LIN {X 0,Y 573.745,Z 549.18,A -85,B 0,C 180,E1 -2261.974,E2 -2261.974} C_VEL
LIN {X 0,Y 573.825,Z 536.531,A -85,B 0,C 180,E1 -2262.331,E2 -2262.331} C_VEL
LIN {X 0,Y 573.935,Z 523.333,A -85,B 0,C 180,E1 -2262.553,E2 -2262.553} C_VEL
LIN {X 0,Y 573.912,Z 426.198,A -85,B 0,C 180,E1 -2263.777,E2 -2263.777} C_VEL
LIN {X 0,Y 573.403,Z 422.615,A -85,B 0,C 180,E1 -2263.85,E2 -2263.85} C_VEL
LIN {X 0,Y 573.571,Z 402.121,A -85,B 0,C 180,E1 -2266.727,E2 -2266.727} C_VEL
LIN {X 0,Y 573.815,Z 381.614,A -85,B 0,C 180,E1 -2269.645,E2 -2269.645} C_VEL
LIN {X 0,Y 574.108,Z 361.938,A -85,B 0,C 180,E1 -2272.491,E2 -2272.491} C_VEL
LIN {X 0,Y 573.627,Z 356.944,A -85,B 0,C 180,E1 -2273.235,E2 -2273.235} C_VEL
LIN {X 0,Y 573.261,Z 355.081,A -85,B 0,C 180,E1 -2273.543,E2 -2273.543} C_VEL
LIN {X 0,Y 573.265,Z 355.076,A -85,B 0,C 180,E1 -2276.189,E2 -2276.189} C_VEL
LIN {X 0,Y 573.239,Z 355.076,A -85,B 0,C 180,E1 -2278.564,E2 -2278.564} C_VEL
LIN {X 0,Y 573.235,Z 355.076,A -85,B 0,C 180,E1 -2280.992,E2 -2280.992} C_VEL
LIN {X 0,Y 573.261,Z 355.078,A -85,B 0,C 180,E1 -2283.523,E2 -2283.523} C_VEL
LIN {X 0,Y 573.26,Z 355.076,A -85,B 0,C 180,E1 -2286.047,E2 -2286.047} C_VEL
LIN {X 0,Y 573.247,Z 355.073,A -85,B 0,C 180,E1 -2288.7,E2 -2288.7} C_VEL
LIN {X 0,Y 573.251,Z 355.083,A -85,B 0,C 180,E1 -2291.595,E2 -2291.595} C_VEL
LIN {X 0,Y 573.235,Z 355.075,A -85,B 0,C 180,E1 -2294.332,E2 -2294.332} C_VEL
LIN {X 0,Y 573.247,Z 355.08,A -85,B 0,C 180,E1 -2297.356,E2 -2297.356} C_VEL
LIN {X 0,Y 573.245,Z 355.073,A -85,B 0,C 180,E1 -2300.393,E2 -2300.393} C_VEL
LIN {X 0,Y 573.251,Z 355.077,A -85,B 0,C 180,E1 -2303.077,E2 -2303.077} C_VEL
LIN {X 0,Y 573.268,Z 355.076,A -85,B 0,C 180,E1 -2305.671,E2 -2305.671} C_VEL
LIN {X 0,Y 573.245,Z 355.074,A -85,B 0,C 180,E1 -2308.185,E2 -2308.185} C_VEL
LIN {X 0,Y 573.264,Z 355.072,A -85,B 0,C 180,E1 -2310.634,E2 -2310.634} C_VEL
LIN {X 0,Y 573.265,Z 355.078,A -85,B 0,C 180,E1 -2313.499,E2 -2313.499} C_VEL
LIN {X 0,Y 573.237,Z 355.074,A -85,B 0,C 180,E1 -2316.135,E2 -2316.135} C_VEL
LIN {X 0,Y 573.252,Z 355.075,A -85,B 0,C 180,E1 -2318.706,E2 -2318.706} C_VEL
LIN {X 0,Y 573.233,Z 355.081,A -85,B 0,C 180,E1 -2321.412,E2 -2321.412} C_VEL
LIN {X 0,Y 573.253,Z 355.075,A -85,B 0,C 180,E1 -2323.622,E2 -2323.622} C_VEL
LIN {X 0,Y 573.232,Z 355.077,A -85,B 0,C 180,E1 -2326.529,E2 -2326.529} C_VEL
LIN {X 0,Y 573.269,Z 355.075,A -85,B 0,C 180,E1 -2329.403,E2 -2329.403} C_VEL
LIN {X 0,Y 573.282,Z 355.069,A -85,B 0,C 180,E1 -2332.25,E2 -2332.25} C_VEL
LIN {X 0,Y 573.308,Z 355.075,A -85,B 0,C 180,E1 -2335.077,E2 -2335.077} C_VEL
LIN {X 0,Y 573.301,Z 355.066,A -85,B 0,C 180,E1 -2337.892,E2 -2337.892} C_VEL
LIN {X 0,Y 573.333,Z 355.069,A -85,B 0,C 180,E1 -2340.702,E2 -2340.702} C_VEL
LIN {X 0,Y 573.238,Z 355.076,A -85,B 0,C 180,E1 -2343.515,E2 -2343.515} C_VEL
LIN {X 0,Y 573.287,Z 355.069,A -85,B 0,C 180,E1 -2345.628,E2 -2345.628} C_VEL
LIN {X 0,Y 573.3,Z 355.071,A -85,B 0,C 180,E1 -2348.459,E2 -2348.459} C_VEL
LIN {X 0,Y 573.29,Z 355.07,A -85,B 0,C 180,E1 -2351.312,E2 -2351.312} C_VEL
LIN {X 0,Y 573.272,Z 355.075,A -85,B 0,C 180,E1 -2354.425,E2 -2354.425} C_VEL
LIN {X 0,Y 573.253,Z 355.076,A -85,B 0,C 180,E1 -2357.112,E2 -2357.112} C_VEL
LIN {X 0,Y 573.251,Z 355.074,A -85,B 0,C 180,E1 -2360.077,E2 -2360.077} C_VEL
LIN {X 0,Y 573.264,Z 355.073,A -85,B 0,C 180,E1 -2363.154,E2 -2363.154} C_VEL
LIN {X 0,Y 573.247,Z 355.079,A -85,B 0,C 180,E1 -2364.408,E2 -2364.408} C_VEL
LIN {X 0,Y 572.616,Z 355.163,A -85,B 0,C 180,E1 -2364.994,E2 -2364.994} C_VEL
LIN {X 0,Y 569.776,Z 355.516,A -85,B 0,C 180,E1 -2365.946,E2 -2365.946} C_VEL
LIN {X 0,Y 567.349,Z 355.816,A -85,B 0,C 180,E1 -2366.712,E2 -2366.712} C_VEL
LIN {X 0,Y 566.298,Z 355.94,A -85,B 0,C 180,E1 -2367.303,E2 -2367.303} C_VEL
LIN {X 0,Y 566.21,Z 355.95,A -85,B 0,C 180,E1 -2367.503,E2 -2367.503} C_VEL
LIN {X 0,Y 566.182,Z 355.962,A -85,B 0,C 180,E1 -2370.593,E2 -2370.593} C_VEL
LIN {X 0,Y 566.223,Z 355.95,A -85,B 0,C 180,E1 -2373.102,E2 -2373.102} C_VEL
LIN {X 0,Y 566.2,Z 355.957,A -85,B 0,C 180,E1 -2376.216,E2 -2376.216} C_VEL
LIN {X 0,Y 566.216,Z 355.949,A -85,B 0,C 180,E1 -2379.274,E2 -2379.274} C_VEL
LIN {X 0,Y 566.212,Z 355.955,A -85,B 0,C 180,E1 -2382.088,E2 -2382.088} C_VEL
LIN {X 0,Y 566.169,Z 355.956,A -85,B 0,C 180,E1 -2385.037,E2 -2385.037} C_VEL
LIN {X 0,Y 566.186,Z 355.957,A -85,B 0,C 180,E1 -2387.911,E2 -2387.911} C_VEL
LIN {X 0,Y 566.22,Z 355.951,A -85,B 0,C 180,E1 -2390.728,E2 -2390.728} C_VEL
LIN {X 0,Y 566.217,Z 355.952,A -85,B 0,C 180,E1 -2393.784,E2 -2393.784} C_VEL
LIN {X 0,Y 566.212,Z 355.958,A -85,B 0,C 180,E1 -2396.266,E2 -2396.266} C_VEL
LIN {X 0,Y 566.198,Z 355.952,A -85,B 0,C 180,E1 -2398.923,E2 -2398.923} C_VEL
LIN {X 0,Y 566.212,Z 355.955,A -85,B 0,C 180,E1 -2401.858,E2 -2401.858} C_VEL
LIN {X 0,Y 566.215,Z 355.957,A -85,B 0,C 180,E1 -2404.252,E2 -2404.252} C_VEL
LIN {X 0,Y 566.171,Z 355.957,A -85,B 0,C 180,E1 -2406.72,E2 -2406.72} C_VEL
LIN {X 0,Y 566.209,Z 355.956,A -85,B 0,C 180,E1 -2409.663,E2 -2409.663} C_VEL
LIN {X 0,Y 566.264,Z 356.15,A -85,B 0,C 180,E1 -2410.878,E2 -2410.878} C_VEL
LIN {X 0,Y 566.436,Z 363.825,A -85,B 0,C 180,E1 -2412.304,E2 -2412.304} C_VEL
LIN {X 0,Y 566.321,Z 379.961,A -85,B 0,C 180,E1 -2415.249,E2 -2415.249} C_VEL
LIN {X 0,Y 566.257,Z 384.42,A -85,B 0,C 180,E1 -2416.055,E2 -2416.055} C_VEL
LIN {X 0,Y 567.176,Z 390.378,A -85,B 0,C 180,E1 -2416.155,E2 -2416.155} C_VEL
LIN {X 0,Y 566.94,Z 490.984,A -85,B 0,C 180,E1 -2417.448,E2 -2417.448} C_VEL
LIN {X 0,Y 566.86,Z 504.235,A -85,B 0,C 180,E1 -2417.765,E2 -2417.765} C_VEL
LIN {X 0,Y 566.745,Z 516.388,A -85,B 0,C 180,E1 -2418.194,E2 -2418.194} C_VEL
LIN {X 0,Y 566.619,Z 528.384,A -85,B 0,C 180,E1 -2418.766,E2 -2418.766} C_VEL
LIN {X 0,Y 566.464,Z 539.56,A -85,B 0,C 180,E1 -2419.456,E2 -2419.456} C_VEL
LIN {X 0,Y 566.326,Z 550.076,A -85,B 0,C 180,E1 -2420.266,E2 -2420.266} C_VEL
LIN {X 0,Y 566.221,Z 558.671,A -85,B 0,C 180,E1 -2421.075,E2 -2421.075} C_VEL
LIN {X 0,Y 566.113,Z 566.592,A -85,B 0,C 180,E1 -2421.972,E2 -2421.972} C_VEL
LIN {X 0,Y 566.05,Z 573.16,A -85,B 0,C 180,E1 -2422.868,E2 -2422.868} C_VEL
LIN {X 0,Y 566.003,Z 579.628,A -85,B 0,C 180,E1 -2423.942,E2 -2423.942} C_VEL
LIN {X 0,Y 565.878,Z 584.765,A -85,B 0,C 180,E1 -2425.013,E2 -2425.013} C_VEL
LIN {X 0,Y 565.926,Z 588.754,A -85,B 0,C 180,E1 -2426.084,E2 -2426.084} C_VEL
LIN {X 0,Y 565.877,Z 591.702,A -85,B 0,C 180,E1 -2427.153,E2 -2427.153} C_VEL
LIN {X 0,Y 565.84,Z 593.128,A -85,B 0,C 180,E1 -2427.865,E2 -2427.865} C_VEL
LIN {X 0,Y 565.841,Z 594.756,A -85,B 0,C 180,E1 -2429.288,E2 -2429.288} C_VEL
LIN {X 0,Y 565.839,Z 594.996,A -85,B 0,C 180,E1 -2430,E2 -2430} C_VEL
LIN {X 0,Y 565.841,Z 594.815,A -85,B 0,C 180,E1 -2430.712,E2 -2430.712} C_VEL
LIN {X 0,Y 565.841,Z 593.268,A -85,B 0,C 180,E1 -2432.135,E2 -2432.135} C_VEL
LIN {X 0,Y 565.878,Z 591.907,A -85,B 0,C 180,E1 -2432.847,E2 -2432.847} C_VEL
LIN {X 0,Y 565.927,Z 589.03,A -85,B 0,C 180,E1 -2433.916,E2 -2433.916} C_VEL
LIN {X 0,Y 565.878,Z 585.13,A -85,B 0,C 180,E1 -2434.987,E2 -2434.987} C_VEL
LIN {X 0,Y 565.99,Z 580.097,A -85,B 0,C 180,E1 -2436.058,E2 -2436.058} C_VEL
LIN {X 0,Y 566.031,Z 573.773,A -85,B 0,C 180,E1 -2437.132,E2 -2437.132} C_VEL
LIN {X 0,Y 566.128,Z 565.852,A -85,B 0,C 180,E1 -2438.208,E2 -2438.208} C_VEL
LIN {X 0,Y 566.249,Z 556.001,A -85,B 0,C 180,E1 -2439.285,E2 -2439.285} C_VEL
LIN {X 0,Y 566.42,Z 545.683,A -85,B 0,C 180,E1 -2440.184,E2 -2440.184} C_VEL
LIN {X 0,Y 566.56,Z 534.375,A -85,B 0,C 180,E1 -2440.973,E2 -2440.973} C_VEL
LIN {X 0,Y 566.691,Z 523.193,A -85,B 0,C 180,E1 -2441.592,E2 -2441.592} C_VEL
LIN {X 0,Y 566.794,Z 510.602,A -85,B 0,C 180,E1 -2442.119,E2 -2442.119} C_VEL
LIN {X 0,Y 566.876,Z 497.43,A -85,B 0,C 180,E1 -2442.508,E2 -2442.508} C_VEL
LIN {X 0,Y 566.978,Z 485.069,A -85,B 0,C 180,E1 -2442.733,E2 -2442.733} C_VEL
LIN {X 0,Y 567.07,Z 389.372,A -85,B 0,C 180,E1 -2443.951,E2 -2443.951} C_VEL
LIN {X 0,Y 566.252,Z 384.332,A -85,B 0,C 180,E1 -2444.051,E2 -2444.051} C_VEL
LIN {X 0,Y 566.417,Z 367.153,A -85,B 0,C 180,E1 -2447.175,E2 -2447.175} C_VEL
LIN {X 0,Y 566.346,Z 356.612,A -85,B 0,C 180,E1 -2449.123,E2 -2449.123} C_VEL
LIN {X 0,Y 566.235,Z 355.953,A -85,B 0,C 180,E1 -2449.295,E2 -2449.295} C_VEL
LIN {X 0,Y 566.197,Z 355.961,A -85,B 0,C 180,E1 -2451.862,E2 -2451.862} C_VEL
LIN {X 0,Y 566.238,Z 355.948,A -85,B 0,C 180,E1 -2454.96,E2 -2454.96} C_VEL
LIN {X 0,Y 566.212,Z 355.951,A -85,B 0,C 180,E1 -2457.338,E2 -2457.338} C_VEL
LIN {X 0,Y 566.203,Z 355.957,A -85,B 0,C 180,E1 -2459.768,E2 -2459.768} C_VEL
LIN {X 0,Y 566.206,Z 355.953,A -85,B 0,C 180,E1 -2462.43,E2 -2462.43} C_VEL
LIN {X 0,Y 566.213,Z 355.949,A -85,B 0,C 180,E1 -2464.994,E2 -2464.994} C_VEL
LIN {X 0,Y 566.195,Z 355.955,A -85,B 0,C 180,E1 -2467.46,E2 -2467.46} C_VEL
LIN {X 0,Y 566.225,Z 355.952,A -85,B 0,C 180,E1 -2470.196,E2 -2470.196} C_VEL
LIN {X 0,Y 566.197,Z 355.952,A -85,B 0,C 180,E1 -2473.053,E2 -2473.053} C_VEL
LIN {X 0,Y 566.198,Z 355.956,A -85,B 0,C 180,E1 -2476.047,E2 -2476.047} C_VEL
LIN {X 0,Y 566.207,Z 355.95,A -85,B 0,C 180,E1 -2478.863,E2 -2478.863} C_VEL
LIN {X 0,Y 566.185,Z 355.963,A -85,B 0,C 180,E1 -2481.637,E2 -2481.637} C_VEL
LIN {X 0,Y 566.206,Z 355.951,A -85,B 0,C 180,E1 -2484.311,E2 -2484.311} C_VEL
LIN {X 0,Y 566.223,Z 355.949,A -85,B 0,C 180,E1 -2486.898,E2 -2486.898} C_VEL
LIN {X 0,Y 566.182,Z 355.961,A -85,B 0,C 180,E1 -2489.407,E2 -2489.407} C_VEL
LIN {X 0,Y 566.221,Z 355.953,A -85,B 0,C 180,E1 -2491.858,E2 -2491.858} C_VEL
LIN {X 0,Y 566.217,Z 355.949,A -85,B 0,C 180,E1 -2494.251,E2 -2494.251} C_VEL
LIN {X 0,Y 566.196,Z 355.961,A -85,B 0,C 180,E1 -2497.369,E2 -2497.369} C_VEL
LIN {X 0,Y 566.213,Z 355.955,A -85,B 0,C 180,E1 -2499.663,E2 -2499.663} C_VEL
LIN {X 0,Y 566.197,Z 355.952,A -85,B 0,C 180,E1 -2502.668,E2 -2502.668} C_VEL
LIN {X 0,Y 566.224,Z 355.953,A -85,B 0,C 180,E1 -2505.626,E2 -2505.626} C_VEL
LIN {X 0,Y 566.266,Z 355.944,A -85,B 0,C 180,E1 -2508.654,E2 -2508.654} C_VEL
LIN {X 0,Y 566.241,Z 355.952,A -85,B 0,C 180,E1 -2511.434,E2 -2511.434} C_VEL
LIN {X 0,Y 566.254,Z 355.944,A -85,B 0,C 180,E1 -2514.302,E2 -2514.302} C_VEL
LIN {X 0,Y 566.273,Z 355.943,A -85,B 0,C 180,E1 -2517.866,E2 -2517.866} C_VEL
LIN {X 0,Y 566.301,Z 355.942,A -85,B 0,C 180,E1 -2520.711,E2 -2520.711} C_VEL
LIN {X 0,Y 566.274,Z 355.948,A -85,B 0,C 180,E1 -2522.846,E2 -2522.846} C_VEL
LIN {X 0,Y 566.255,Z 355.945,A -85,B 0,C 180,E1 -2525.698,E2 -2525.698} C_VEL
LIN {X 0,Y 566.242,Z 355.949,A -85,B 0,C 180,E1 -2528.565,E2 -2528.565} C_VEL
LIN {X 0,Y 566.242,Z 355.948,A -85,B 0,C 180,E1 -2531.454,E2 -2531.454} C_VEL
LIN {X 0,Y 566.225,Z 355.952,A -85,B 0,C 180,E1 -2534.507,E2 -2534.507} C_VEL
LIN {X 0,Y 566.197,Z 355.954,A -85,B 0,C 180,E1 -2537.332,E2 -2537.332} C_VEL
LIN {X 0,Y 566.216,Z 355.952,A -85,B 0,C 180,E1 -2540.337,E2 -2540.337} C_VEL
LIN {X 0,Y 566.222,Z 355.95,A -85,B 0,C 180,E1 -2543.402,E2 -2543.402} C_VEL
LIN {X 0,Y 566.218,Z 355.949,A -85,B 0,C 180,E1 -2545.749,E2 -2545.749} C_VEL
LIN {X 0,Y 566.202,Z 355.953,A -85,B 0,C 180,E1 -2548.204,E2 -2548.204} C_VEL
LIN {X 0,Y 566.194,Z 355.955,A -85,B 0,C 180,E1 -2551.079,E2 -2551.079} C_VEL
LIN {X 0,Y 566.223,Z 355.948,A -85,B 0,C 180,E1 -2553.738,E2 -2553.738} C_VEL
LIN {X 0,Y 566.211,Z 355.96,A -85,B 0,C 180,E1 -2556.569,E2 -2556.569} C_VEL
LIN {X 0,Y 566.209,Z 355.95,A -85,B 0,C 180,E1 -2559.687,E2 -2559.687} C_VEL
LIN {X 0,Y 566.213,Z 355.953,A -85,B 0,C 180,E1 -2562.088,E2 -2562.088} C_VEL
LIN {X 0,Y 566.17,Z 355.957,A -85,B 0,C 180,E1 -2565.036,E2 -2565.036} C_VEL
LIN {X 0,Y 566.215,Z 355.954,A -85,B 0,C 180,E1 -2568.137,E2 -2568.137} C_VEL
LIN {X 0,Y 566.22,Z 355.953,A -85,B 0,C 180,E1 -2570.728,E2 -2570.728} C_VEL
LIN {X 0,Y 566.217,Z 355.951,A -85,B 0,C 180,E1 -2573.784,E2 -2573.784} C_VEL
LIN {X 0,Y 566.211,Z 355.959,A -85,B 0,C 180,E1 -2576.266,E2 -2576.266} C_VEL
LIN {X 0,Y 566.198,Z 355.952,A -85,B 0,C 180,E1 -2578.923,E2 -2578.923} C_VEL
LIN {X 0,Y 566.211,Z 355.955,A -85,B 0,C 180,E1 -2581.858,E2 -2581.858} C_VEL
LIN {X 0,Y 566.215,Z 355.959,A -85,B 0,C 180,E1 -2584.252,E2 -2584.252} C_VEL
LIN {X 0,Y 566.236,Z 356.138,A -85,B 0,C 180,E1 -2586.356,E2 -2586.356} C_VEL
LIN {X 0,Y 567.11,Z 361.752,A -85,B 0,C 180,E1 -2587.216,E2 -2587.216} C_VEL
LIN {X 0,Y 566.912,Z 380.06,A -85,B 0,C 180,E1 -2589.879,E2 -2589.879} C_VEL
LIN {X 0,Y 566.61,Z 400.895,A -85,B 0,C 180,E1 -2592.885,E2 -2592.885} C_VEL
LIN {X 0,Y 566.403,Z 422.615,A -85,B 0,C 180,E1 -2595.975,E2 -2595.975} C_VEL
LIN {X 0,Y 567.22,Z 429.316,A -85,B 0,C 180,E1 -2596.097,E2 -2596.097} C_VEL
LIN {X 0,Y 566.937,Z 530.961,A -85,B 0,C 180,E1 -2597.403,E2 -2597.403} C_VEL
LIN {X 0,Y 566.859,Z 544.228,A -85,B 0,C 180,E1 -2597.719,E2 -2597.719} C_VEL
LIN {X 0,Y 566.758,Z 556.383,A -85,B 0,C 180,E1 -2598.149,E2 -2598.149} C_VEL
LIN {X 0,Y 566.589,Z 568.447,A -85,B 0,C 180,E1 -2598.724,E2 -2598.724} C_VEL
LIN {X 0,Y 566.442,Z 580.203,A -85,B 0,C 180,E1 -2599.455,E2 -2599.455} C_VEL
LIN {X 0,Y 566.321,Z 590.605,A -85,B 0,C 180,E1 -2600.266,E2 -2600.266} C_VEL
LIN {X 0,Y 566.207,Z 599.115,A -85,B 0,C 180,E1 -2601.074,E2 -2601.074} C_VEL
LIN {X 0,Y 566.112,Z 606.962,A -85,B 0,C 180,E1 -2601.972,E2 -2601.972} C_VEL
LIN {X 0,Y 566.003,Z 614.623,A -85,B 0,C 180,E1 -2603.047,E2 -2603.047} C_VEL
LIN {X 0,Y 566.004,Z 621.68,A -85,B 0,C 180,E1 -2604.299,E2 -2604.299} C_VEL
LIN {X 0,Y 565.933,Z 626.373,A -85,B 0,C 180,E1 -2605.37,E2 -2605.37} C_VEL
LIN {X 0,Y 565.927,Z 629.958,A -85,B 0,C 180,E1 -2606.44,E2 -2606.44} C_VEL
LIN {X 0,Y 565.878,Z 631.808,A -85,B 0,C 180,E1 -2607.153,E2 -2607.153} C_VEL
LIN {X 0,Y 565.846,Z 634.185,A -85,B 0,C 180,E1 -2608.577,E2 -2608.577} C_VEL
LIN {X 0,Y 565.839,Z 635,A -85,B 0,C 180,E1 -2610,E2 -2610} C_VEL
LIN {X 0,Y 565.846,Z 634.186,A -85,B 0,C 180,E1 -2611.423,E2 -2611.423} C_VEL
LIN {X 0,Y 565.878,Z 631.81,A -85,B 0,C 180,E1 -2612.847,E2 -2612.847} C_VEL
LIN {X 0,Y 565.926,Z 628.896,A -85,B 0,C 180,E1 -2613.916,E2 -2613.916} C_VEL
LIN {X 0,Y 565.878,Z 624.949,A -85,B 0,C 180,E1 -2614.987,E2 -2614.987} C_VEL
LIN {X 0,Y 566.002,Z 619.868,A -85,B 0,C 180,E1 -2616.058,E2 -2616.058} C_VEL
LIN {X 0,Y 566.04,Z 613.469,A -85,B 0,C 180,E1 -2617.132,E2 -2617.132} C_VEL
LIN {X 0,Y 566.133,Z 605.479,A -85,B 0,C 180,E1 -2618.207,E2 -2618.207} C_VEL
LIN {X 0,Y 566.228,Z 597.337,A -85,B 0,C 180,E1 -2619.105,E2 -2619.105} C_VEL
LIN {X 0,Y 566.343,Z 587.403,A -85,B 0,C 180,E1 -2620.005,E2 -2620.005} C_VEL
LIN {X 0,Y 566.529,Z 576.294,A -85,B 0,C 180,E1 -2620.807,E2 -2620.807} C_VEL
LIN {X 0,Y 566.612,Z 565.181,A -85,B 0,C 180,E1 -2621.446,E2 -2621.446} C_VEL
LIN {X 0,Y 566.736,Z 552.989,A -85,B 0,C 180,E1 -2621.988,E2 -2621.988} C_VEL
LIN {X 0,Y 566.892,Z 540.187,A -85,B 0,C 180,E1 -2622.394,E2 -2622.394} C_VEL
LIN {X 0,Y 567.001,Z 528.125,A -85,B 0,C 180,E1 -2622.641,E2 -2622.641} C_VEL
LIN {X 0,Y 567.055,Z 427.203,A -85,B 0,C 180,E1 -2623.934,E2 -2623.934} C_VEL
LIN {X 0,Y 566.403,Z 422.615,A -85,B 0,C 180,E1 -2624.025,E2 -2624.025} C_VEL
LIN {X 0,Y 566.61,Z 400.895,A -85,B 0,C 180,E1 -2627.115,E2 -2627.115} C_VEL
LIN {X 0,Y 566.912,Z 380.062,A -85,B 0,C 180,E1 -2630.121,E2 -2630.121} C_VEL
LIN {X 0,Y 567.109,Z 361.752,A -85,B 0,C 180,E1 -2632.784,E2 -2632.784} C_VEL
LIN {X 0,Y 566.22,Z 355.959,A -85,B 0,C 180,E1 -2633.693,E2 -2633.693} C_VEL
LIN {X 0,Y 566.216,Z 355.95,A -85,B 0,C 180,E1 -2636.54,E2 -2636.54} C_VEL
LIN {X 0,Y 566.193,Z 355.953,A -85,B 0,C 180,E1 -2638.953,E2 -2638.953} C_VEL
LIN {X 0,Y 566.2,Z 355.957,A -85,B 0,C 180,E1 -2641.421,E2 -2641.421} C_VEL
LIN {X 0,Y 566.212,Z 355.955,A -85,B 0,C 180,E1 -2643.955,E2 -2643.955} C_VEL
LIN {X 0,Y 566.215,Z 355.949,A -85,B 0,C 180,E1 -2646.568,E2 -2646.568} C_VEL
LIN {X 0,Y 566.211,Z 355.959,A -85,B 0,C 180,E1 -2649.685,E2 -2649.685} C_VEL
LIN {X 0,Y 566.211,Z 355.952,A -85,B 0,C 180,E1 -2652.086,E2 -2652.086} C_VEL
LIN {X 0,Y 566.17,Z 355.957,A -85,B 0,C 180,E1 -2655.035,E2 -2655.035} C_VEL
LIN {X 0,Y 566.213,Z 355.953,A -85,B 0,C 180,E1 -2657.912,E2 -2657.912} C_VEL
LIN {X 0,Y 566.218,Z 355.949,A -85,B 0,C 180,E1 -2660.726,E2 -2660.726} C_VEL
LIN {X 0,Y 566.212,Z 355.954,A -85,B 0,C 180,E1 -2663.783,E2 -2663.783} C_VEL
LIN {X 0,Y 566.223,Z 355.948,A -85,B 0,C 180,E1 -2666.262,E2 -2666.262} C_VEL
LIN {X 0,Y 566.197,Z 355.954,A -85,B 0,C 180,E1 -2668.921,E2 -2668.921} C_VEL
LIN {X 0,Y 566.192,Z 355.957,A -85,B 0,C 180,E1 -2671.047,E2 -2671.047} C_VEL
LIN {X 0,Y 566.24,Z 355.953,A -85,B 0,C 180,E1 -2673.46,E2 -2673.46} C_VEL
LIN {X 0,Y 566.197,Z 355.953,A -85,B 0,C 180,E1 -2675.819,E2 -2675.819} C_VEL
LIN {X 0,Y 566.211,Z 355.954,A -85,B 0,C 180,E1 -2678.902,E2 -2678.902} C_VEL
LIN {X 0,Y 566.206,Z 355.96,A -85,B 0,C 180,E1 -2681.172,E2 -2681.172} C_VEL
LIN {X 0,Y 566.215,Z 355.955,A -85,B 0,C 180,E1 -2683.412,E2 -2683.412} C_VEL
LIN {X 0,Y 566.194,Z 355.952,A -85,B 0,C 180,E1 -2686.359,E2 -2686.359} C_VEL
LIN {X 0,Y 566.266,Z 355.946,A -85,B 0,C 180,E1 -2688.654,E2 -2688.654} C_VEL
LIN {X 0,Y 566.241,Z 355.95,A -85,B 0,C 180,E1 -2691.434,E2 -2691.434} C_VEL
LIN {X 0,Y 566.255,Z 355.945,A -85,B 0,C 180,E1 -2694.302,E2 -2694.302} C_VEL
LIN {X 0,Y 566.273,Z 355.942,A -85,B 0,C 180,E1 -2697.866,E2 -2697.866} C_VEL
LIN {X 0,Y 566.303,Z 355.944,A -85,B 0,C 180,E1 -2700.711,E2 -2700.711} C_VEL
LIN {X 0,Y 566.274,Z 355.951,A -85,B 0,C 180,E1 -2702.846,E2 -2702.846} C_VEL
LIN {X 0,Y 566.255,Z 355.944,A -85,B 0,C 180,E1 -2705.698,E2 -2705.698} C_VEL
LIN {X 0,Y 566.241,Z 355.951,A -85,B 0,C 180,E1 -2708.566,E2 -2708.566} C_VEL
LIN {X 0,Y 566.242,Z 355.947,A -85,B 0,C 180,E1 -2711.454,E2 -2711.454} C_VEL
LIN {X 0,Y 566.225,Z 355.954,A -85,B 0,C 180,E1 -2714.507,E2 -2714.507} C_VEL
LIN {X 0,Y 566.197,Z 355.953,A -85,B 0,C 180,E1 -2717.332,E2 -2717.332} C_VEL
LIN {X 0,Y 566.213,Z 355.954,A -85,B 0,C 180,E1 -2720.337,E2 -2720.337} C_VEL
LIN {X 0,Y 566.222,Z 355.949,A -85,B 0,C 180,E1 -2723.403,E2 -2723.403} C_VEL
LIN {X 0,Y 566.218,Z 355.949,A -85,B 0,C 180,E1 -2725.749,E2 -2725.749} C_VEL
LIN {X 0,Y 566.21,Z 355.95,A -85,B 0,C 180,E1 -2727.503,E2 -2727.503} C_VEL
LIN {X 0,Y 565.53,Z 356.039,A -85,B 0,C 180,E1 -2728.097,E2 -2728.097} C_VEL
LIN {X 0,Y 562.659,Z 356.394,A -85,B 0,C 180,E1 -2729.061,E2 -2729.061} C_VEL
LIN {X 0,Y 560.245,Z 356.695,A -85,B 0,C 180,E1 -2729.836,E2 -2729.836} C_VEL
LIN {X 0,Y 559.218,Z 356.829,A -85,B 0,C 180,E1 -2730.435,E2 -2730.435} C_VEL
LIN {X 0,Y 559.139,Z 356.832,A -85,B 0,C 180,E1 -2730.637,E2 -2730.637} C_VEL
LIN {X 0,Y 559.158,Z 356.828,A -85,B 0,C 180,E1 -2733.575,E2 -2733.575} C_VEL
LIN {X 0,Y 559.177,Z 356.836,A -85,B 0,C 180,E1 -2736.451,E2 -2736.451} C_VEL
LIN {X 0,Y 559.173,Z 356.829,A -85,B 0,C 180,E1 -2738.935,E2 -2738.935} C_VEL
LIN {X 0,Y 559.188,Z 356.826,A -85,B 0,C 180,E1 -2741.768,E2 -2741.768} C_VEL
LIN {X 0,Y 559.136,Z 356.834,A -85,B 0,C 180,E1 -2744.74,E2 -2744.74} C_VEL
LIN {X 0,Y 559.154,Z 356.829,A -85,B 0,C 180,E1 -2747.257,E2 -2747.257} C_VEL
LIN {X 0,Y 559.179,Z 356.833,A -85,B 0,C 180,E1 -2750.136,E2 -2750.136} C_VEL
LIN {X 0,Y 559.145,Z 356.831,A -85,B 0,C 180,E1 -2752.893,E2 -2752.893} C_VEL
LIN {X 0,Y 559.156,Z 356.83,A -85,B 0,C 180,E1 -2755.557,E2 -2755.557} C_VEL
LIN {X 0,Y 559.169,Z 356.837,A -85,B 0,C 180,E1 -2758.138,E2 -2758.138} C_VEL
LIN {X 0,Y 559.144,Z 356.832,A -85,B 0,C 180,E1 -2760.647,E2 -2760.647} C_VEL
LIN {X 0,Y 559.171,Z 356.827,A -85,B 0,C 180,E1 -2763.173,E2 -2763.173} C_VEL
LIN {X 0,Y 559.157,Z 356.832,A -85,B 0,C 180,E1 -2765.496,E2 -2765.496} C_VEL
LIN {X 0,Y 559.173,Z 356.83,A -85,B 0,C 180,E1 -2768.624,E2 -2768.624} C_VEL
LIN {X 0,Y 559.235,Z 357.029,A -85,B 0,C 180,E1 -2770.767,E2 -2770.767} C_VEL
LIN {X 0,Y 559.511,Z 363.855,A -85,B 0,C 180,E1 -2772.077,E2 -2772.077} C_VEL
LIN {X 0,Y 559.276,Z 380.241,A -85,B 0,C 180,E1 -2775.109,E2 -2775.109} C_VEL
LIN {X 0,Y 559.214,Z 384.423,A -85,B 0,C 180,E1 -2775.875,E2 -2775.875} C_VEL
LIN {X 0,Y 560.313,Z 391.886,A -85,B 0,C 180,E1 -2776.001,E2 -2776.001} C_VEL
LIN {X 0,Y 560.026,Z 491.013,A -85,B 0,C 180,E1 -2777.291,E2 -2777.291} C_VEL
LIN {X 0,Y 559.917,Z 504.253,A -85,B 0,C 180,E1 -2777.611,E2 -2777.611} C_VEL
LIN {X 0,Y 559.791,Z 516.403,A -85,B 0,C 180,E1 -2778.045,E2 -2778.045} C_VEL
LIN {X 0,Y 559.656,Z 528.029,A -85,B 0,C 180,E1 -2778.604,E2 -2778.604} C_VEL
LIN {X 0,Y 559.476,Z 539.567,A -85,B 0,C 180,E1 -2779.322,E2 -2779.322} C_VEL
LIN {X 0,Y 559.307,Z 550.083,A -85,B 0,C 180,E1 -2780.142,E2 -2780.142} C_VEL
LIN {X 0,Y 559.197,Z 558.677,A -85,B 0,C 180,E1 -2780.962,E2 -2780.962} C_VEL
LIN {X 0,Y 559.05,Z 566.597,A -85,B 0,C 180,E1 -2781.87,E2 -2781.87} C_VEL
LIN {X 0,Y 558.971,Z 574.457,A -85,B 0,C 180,E1 -2782.977,E2 -2782.977} C_VEL
LIN {X 0,Y 558.936,Z 581.455,A -85,B 0,C 180,E1 -2784.227,E2 -2784.227} C_VEL
LIN {X 0,Y 558.827,Z 586.195,A -85,B 0,C 180,E1 -2785.311,E2 -2785.311} C_VEL
LIN {X 0,Y 558.836,Z 589.828,A -85,B 0,C 180,E1 -2786.395,E2 -2786.395} C_VEL
LIN {X 0,Y 558.799,Z 591.704,A -85,B 0,C 180,E1 -2787.116,E2 -2787.116} C_VEL
LIN {X 0,Y 558.746,Z 593.128,A -85,B 0,C 180,E1 -2787.838,E2 -2787.838} C_VEL
LIN {X 0,Y 558.741,Z 594.757,A -85,B 0,C 180,E1 -2789.279,E2 -2789.279} C_VEL
LIN {X 0,Y 558.74,Z 594.996,A -85,B 0,C 180,E1 -2790,E2 -2790} C_VEL
LIN {X 0,Y 558.741,Z 594.815,A -85,B 0,C 180,E1 -2790.721,E2 -2790.721} C_VEL
LIN {X 0,Y 558.746,Z 593.266,A -85,B 0,C 180,E1 -2792.162,E2 -2792.162} C_VEL
LIN {X 0,Y 558.8,Z 591.905,A -85,B 0,C 180,E1 -2792.884,E2 -2792.884} C_VEL
LIN {X 0,Y 558.844,Z 589.028,A -85,B 0,C 180,E1 -2793.966,E2 -2793.966} C_VEL
LIN {X 0,Y 558.798,Z 585.127,A -85,B 0,C 180,E1 -2795.051,E2 -2795.051} C_VEL
LIN {X 0,Y 558.91,Z 580.095,A -85,B 0,C 180,E1 -2796.136,E2 -2796.136} C_VEL
LIN {X 0,Y 558.972,Z 573.769,A -85,B 0,C 180,E1 -2797.223,E2 -2797.223} C_VEL
LIN {X 0,Y 559.091,Z 565.847,A -85,B 0,C 180,E1 -2798.312,E2 -2798.312} C_VEL
LIN {X 0,Y 559.223,Z 555.994,A -85,B 0,C 180,E1 -2799.403,E2 -2799.403} C_VEL
LIN {X 0,Y 559.412,Z 545.676,A -85,B 0,C 180,E1 -2800.313,E2 -2800.313} C_VEL
LIN {X 0,Y 559.585,Z 534.697,A -85,B 0,C 180,E1 -2801.09,E2 -2801.09} C_VEL
LIN {X 0,Y 559.711,Z 524.458,A -85,B 0,C 180,E1 -2801.672,E2 -2801.672} C_VEL
LIN {X 0,Y 559.818,Z 512.969,A -85,B 0,C 180,E1 -2802.184,E2 -2802.184} C_VEL
LIN {X 0,Y 559.96,Z 500.153,A -85,B 0,C 180,E1 -2802.595,E2 -2802.595} C_VEL
LIN {X 0,Y 560.073,Z 486.549,A -85,B 0,C 180,E1 -2802.869,E2 -2802.869} C_VEL
LIN {X 0,Y 560.203,Z 390.221,A -85,B 0,C 180,E1 -2804.114,E2 -2804.114} C_VEL
LIN {X 0,Y 559.235,Z 384.329,A -85,B 0,C 180,E1 -2804.231,E2 -2804.231} C_VEL
LIN {X 0,Y 559.4,Z 367.744,A -85,B 0,C 180,E1 -2807.287,E2 -2807.287} C_VEL
LIN {X 0,Y 559.401,Z 358.347,A -85,B 0,C 180,E1 -2809.065,E2 -2809.065} C_VEL
LIN {X 0,Y 559.19,Z 356.832,A -85,B 0,C 180,E1 -2809.412,E2 -2809.412} C_VEL
LIN {X 0,Y 559.144,Z 356.841,A -85,B 0,C 180,E1 -2812.152,E2 -2812.152} C_VEL
LIN {X 0,Y 559.181,Z 356.828,A -85,B 0,C 180,E1 -2815.186,E2 -2815.186} C_VEL
LIN {X 0,Y 559.182,Z 356.831,A -85,B 0,C 180,E1 -2817.711,E2 -2817.711} C_VEL
LIN {X 0,Y 559.157,Z 356.834,A -85,B 0,C 180,E1 -2820.182,E2 -2820.182} C_VEL
LIN {X 0,Y 559.175,Z 356.826,A -85,B 0,C 180,E1 -2822.713,E2 -2822.713} C_VEL
LIN {X 0,Y 559.157,Z 356.83,A -85,B 0,C 180,E1 -2825.321,E2 -2825.321} C_VEL
LIN {X 0,Y 559.133,Z 356.838,A -85,B 0,C 180,E1 -2828.017,E2 -2828.017} C_VEL
LIN {X 0,Y 559.17,Z 356.827,A -85,B 0,C 180,E1 -2830.81,E2 -2830.81} C_VEL
LIN {X 0,Y 559.155,Z 356.838,A -85,B 0,C 180,E1 -2833.731,E2 -2833.731} C_VEL
LIN {X 0,Y 559.164,Z 356.827,A -85,B 0,C 180,E1 -2836.8,E2 -2836.8} C_VEL
LIN {X 0,Y 559.172,Z 356.829,A -85,B 0,C 180,E1 -2839.189,E2 -2839.189} C_VEL
LIN {X 0,Y 559.13,Z 356.836,A -85,B 0,C 180,E1 -2841.982,E2 -2841.982} C_VEL
LIN {X 0,Y 559.151,Z 356.829,A -85,B 0,C 180,E1 -2844.677,E2 -2844.677} C_VEL
LIN {X 0,Y 559.169,Z 356.833,A -85,B 0,C 180,E1 -2847.36,E2 -2847.36} C_VEL
LIN {X 0,Y 559.143,Z 356.832,A -85,B 0,C 180,E1 -2850.141,E2 -2850.141} C_VEL
LIN {X 0,Y 559.172,Z 356.83,A -85,B 0,C 180,E1 -2853.098,E2 -2853.098} C_VEL
LIN {X 0,Y 559.153,Z 356.838,A -85,B 0,C 180,E1 -2855.495,E2 -2855.495} C_VEL
LIN {X 0,Y 559.157,Z 356.828,A -85,B 0,C 180,E1 -2858.447,E2 -2858.447} C_VEL
LIN {X 0,Y 559.164,Z 356.83,A -85,B 0,C 180,E1 -2860.926,E2 -2860.926} C_VEL
LIN {X 0,Y 559.165,Z 356.829,A -85,B 0,C 180,E1 -2863.948,E2 -2863.948} C_VEL
LIN {X 0,Y 559.166,Z 356.827,A -85,B 0,C 180,E1 -2866.184,E2 -2866.184} C_VEL
LIN {X 0,Y 559.203,Z 356.83,A -85,B 0,C 180,E1 -2869.134,E2 -2869.134} C_VEL
LIN {X 0,Y 559.205,Z 356.823,A -85,B 0,C 180,E1 -2872.054,E2 -2872.054} C_VEL
LIN {X 0,Y 559.253,Z 356.823,A -85,B 0,C 180,E1 -2874.953,E2 -2874.953} C_VEL
LIN {X 0,Y 559.244,Z 356.818,A -85,B 0,C 180,E1 -2877.839,E2 -2877.839} C_VEL
LIN {X 0,Y 559.27,Z 356.818,A -85,B 0,C 180,E1 -2880.72,E2 -2880.72} C_VEL
LIN {X 0,Y 559.239,Z 356.825,A -85,B 0,C 180,E1 -2882.881,E2 -2882.881} C_VEL
LIN {X 0,Y 559.224,Z 356.821,A -85,B 0,C 180,E1 -2885.77,E2 -2885.77} C_VEL
LIN {X 0,Y 559.197,Z 356.828,A -85,B 0,C 180,E1 -2888.674,E2 -2888.674} C_VEL
LIN {X 0,Y 559.2,Z 356.824,A -85,B 0,C 180,E1 -2891.601,E2 -2891.601} C_VEL
LIN {X 0,Y 559.19,Z 356.829,A -85,B 0,C 180,E1 -2894.596,E2 -2894.596} C_VEL
LIN {X 0,Y 559.157,Z 356.829,A -85,B 0,C 180,E1 -2897.557,E2 -2897.557} C_VEL
LIN {X 0,Y 559.181,Z 356.832,A -85,B 0,C 180,E1 -2900.605,E2 -2900.605} C_VEL
LIN {X 0,Y 559.159,Z 356.828,A -85,B 0,C 180,E1 -2903.716,E2 -2903.716} C_VEL
LIN {X 0,Y 559.192,Z 356.825,A -85,B 0,C 180,E1 -2906.097,E2 -2906.097} C_VEL
LIN {X 0,Y 559.159,Z 356.835,A -85,B 0,C 180,E1 -2908.53,E2 -2908.53} C_VEL
LIN {X 0,Y 559.148,Z 356.831,A -85,B 0,C 180,E1 -2911.276,E2 -2911.276} C_VEL
LIN {X 0,Y 559.172,Z 356.828,A -85,B 0,C 180,E1 -2913.952,E2 -2913.952} C_VEL
LIN {X 0,Y 559.164,Z 356.835,A -85,B 0,C 180,E1 -2916.449,E2 -2916.449} C_VEL
LIN {X 0,Y 559.173,Z 356.83,A -85,B 0,C 180,E1 -2918.934,E2 -2918.934} C_VEL
LIN {X 0,Y 559.189,Z 356.825,A -85,B 0,C 180,E1 -2921.768,E2 -2921.768} C_VEL
LIN {X 0,Y 559.136,Z 356.836,A -85,B 0,C 180,E1 -2924.74,E2 -2924.74} C_VEL
LIN {X 0,Y 559.16,Z 356.828,A -85,B 0,C 180,E1 -2927.258,E2 -2927.258} C_VEL
LIN {X 0,Y 559.183,Z 356.831,A -85,B 0,C 180,E1 -2930.136,E2 -2930.136} C_VEL
LIN {X 0,Y 559.145,Z 356.832,A -85,B 0,C 180,E1 -2932.893,E2 -2932.893} C_VEL
LIN {X 0,Y 559.157,Z 356.829,A -85,B 0,C 180,E1 -2935.557,E2 -2935.557} C_VEL
LIN {X 0,Y 559.169,Z 356.834,A -85,B 0,C 180,E1 -2938.138,E2 -2938.138} C_VEL
LIN {X 0,Y 559.143,Z 356.835,A -85,B 0,C 180,E1 -2940.647,E2 -2940.647} C_VEL
LIN {X 0,Y 559.171,Z 356.829,A -85,B 0,C 180,E1 -2943.173,E2 -2943.173} C_VEL
LIN {X 0,Y 559.182,Z 356.835,A -85,B 0,C 180,E1 -2946.089,E2 -2946.089} C_VEL
LIN {X 0,Y 559.187,Z 356.91,A -85,B 0,C 180,E1 -2946.187,E2 -2946.187} C_VEL
LIN {X 0,Y 560.168,Z 362.859,A -85,B 0,C 180,E1 -2947.112,E2 -2947.112} C_VEL
LIN {X 0,Y 559.949,Z 381.239,A -85,B 0,C 180,E1 -2949.809,E2 -2949.809} C_VEL
LIN {X 0,Y 559.625,Z 402.635,A -85,B 0,C 180,E1 -2952.918,E2 -2952.918} C_VEL
LIN {X 0,Y 559.406,Z 422.615,A -85,B 0,C 180,E1 -2955.796,E2 -2955.796} C_VEL
LIN {X 0,Y 560.327,Z 430.323,A -85,B 0,C 180,E1 -2955.936,E2 -2955.936} C_VEL
LIN {X 0,Y 560.021,Z 530.961,A -85,B 0,C 180,E1 -2957.245,E2 -2957.245} C_VEL
LIN {X 0,Y 559.941,Z 544.227,A -85,B 0,C 180,E1 -2957.565,E2 -2957.565} C_VEL
LIN {X 0,Y 559.808,Z 556.384,A -85,B 0,C 180,E1 -2957.999,E2 -2957.999} C_VEL
LIN {X 0,Y 559.615,Z 568.321,A -85,B 0,C 180,E1 -2958.574,E2 -2958.574} C_VEL
LIN {X 0,Y 559.461,Z 580.201,A -85,B 0,C 180,E1 -2959.322,E2 -2959.322} C_VEL
LIN {X 0,Y 559.302,Z 590.606,A -85,B 0,C 180,E1 -2960.142,E2 -2960.142} C_VEL
LIN {X 0,Y 559.161,Z 599.115,A -85,B 0,C 180,E1 -2960.961,E2 -2960.961} C_VEL
LIN {X 0,Y 559.05,Z 606.962,A -85,B 0,C 180,E1 -2961.87,E2 -2961.87} C_VEL
LIN {X 0,Y 558.944,Z 614.623,A -85,B 0,C 180,E1 -2962.959,E2 -2962.959} C_VEL
LIN {X 0,Y 558.935,Z 621.68,A -85,B 0,C 180,E1 -2964.227,E2 -2964.227} C_VEL
LIN {X 0,Y 558.827,Z 626.373,A -85,B 0,C 180,E1 -2965.311,E2 -2965.311} C_VEL
LIN {X 0,Y 558.836,Z 629.958,A -85,B 0,C 180,E1 -2966.395,E2 -2966.395} C_VEL
LIN {X 0,Y 558.799,Z 631.808,A -85,B 0,C 180,E1 -2967.116,E2 -2967.116} C_VEL
LIN {X 0,Y 558.745,Z 634.184,A -85,B 0,C 180,E1 -2968.559,E2 -2968.559} C_VEL
LIN {X 0,Y 558.74,Z 635,A -85,B 0,C 180,E1 -2970,E2 -2970} C_VEL
LIN {X 0,Y 558.745,Z 634.185,A -85,B 0,C 180,E1 -2971.441,E2 -2971.441} C_VEL
LIN {X 0,Y 558.799,Z 631.81,A -85,B 0,C 180,E1 -2972.884,E2 -2972.884} C_VEL
LIN {X 0,Y 558.843,Z 628.896,A -85,B 0,C 180,E1 -2973.966,E2 -2973.966} C_VEL
LIN {X 0,Y 558.799,Z 624.949,A -85,B 0,C 180,E1 -2975.051,E2 -2975.051} C_VEL
LIN {X 0,Y 558.921,Z 619.868,A -85,B 0,C 180,E1 -2976.135,E2 -2976.135} C_VEL
LIN {X 0,Y 558.977,Z 613.469,A -85,B 0,C 180,E1 -2977.223,E2 -2977.223} C_VEL
LIN {X 0,Y 559.099,Z 605.479,A -85,B 0,C 180,E1 -2978.311,E2 -2978.311} C_VEL
LIN {X 0,Y 559.184,Z 597.337,A -85,B 0,C 180,E1 -2979.221,E2 -2979.221} C_VEL
LIN {X 0,Y 559.356,Z 587.402,A -85,B 0,C 180,E1 -2980.131,E2 -2980.131} C_VEL
LIN {X 0,Y 559.543,Z 576.403,A -85,B 0,C 180,E1 -2980.937,E2 -2980.937} C_VEL
LIN {X 0,Y 559.671,Z 564.465,A -85,B 0,C 180,E1 -2981.627,E2 -2981.627} C_VEL
LIN {X 0,Y 559.818,Z 551.776,A -85,B 0,C 180,E1 -2982.184,E2 -2982.184} C_VEL
LIN {X 0,Y 559.988,Z 538.358,A -85,B 0,C 180,E1 -2982.595,E2 -2982.595} C_VEL
LIN {X 0,Y 560.076,Z 525.105,A -85,B 0,C 180,E1 -2982.846,E2 -2982.846} C_VEL
LIN {X 0,Y 560.224,Z 428.334,A -85,B 0,C 180,E1 -2984.093,E2 -2984.093} C_VEL
LIN {X 0,Y 559.405,Z 422.615,A -85,B 0,C 180,E1 -2984.204,E2 -2984.204} C_VEL
LIN {X 0,Y 559.652,Z 400.646,A -85,B 0,C 180,E1 -2987.37,E2 -2987.37} C_VEL
LIN {X 0,Y 559.941,Z 379.923,A -85,B 0,C 180,E1 -2990.383,E2 -2990.383} C_VEL
LIN {X 0,Y 560.168,Z 362.847,A -85,B 0,C 180,E1 -2992.888,E2 -2992.888} C_VEL
LIN {X 0,Y 559.179,Z 356.836,A -85,B 0,C 180,E1 -2993.838,E2 -2993.838} C_VEL
LIN {X 0,Y 559.171,Z 356.828,A -85,B 0,C 180,E1 -2996.827,E2 -2996.827} C_VEL
LIN {X 0,Y 559.143,Z 356.835,A -85,B 0,C 180,E1 -2999.353,E2 -2999.353} C_VEL
LIN {X 0,Y 559.169,Z 356.836,A -85,B 0,C 180,E1 -3001.862,E2 -3001.862} C_VEL
LIN {X 0,Y 559.157,Z 356.829,A -85,B 0,C 180,E1 -3004.443,E2 -3004.443} C_VEL
LIN {X 0,Y 559.145,Z 356.832,A -85,B 0,C 180,E1 -3007.107,E2 -3007.107} C_VEL
LIN {X 0,Y 559.167,Z 356.832,A -85,B 0,C 180,E1 -3009.942,E2 -3009.942} C_VEL
LIN {X 0,Y 559.16,Z 356.828,A -85,B 0,C 180,E1 -3012.742,E2 -3012.742} C_VEL
LIN {X 0,Y 559.151,Z 356.835,A -85,B 0,C 180,E1 -3015.76,E2 -3015.76} C_VEL
LIN {X 0,Y 559.189,Z 356.825,A -85,B 0,C 180,E1 -3018.232,E2 -3018.232} C_VEL
LIN {X 0,Y 559.173,Z 356.832,A -85,B 0,C 180,E1 -3021.19,E2 -3021.19} C_VEL
LIN {X 0,Y 559.167,Z 356.831,A -85,B 0,C 180,E1 -3023.791,E2 -3023.791} C_VEL
LIN {X 0,Y 559.171,Z 356.826,A -85,B 0,C 180,E1 -3026.426,E2 -3026.426} C_VEL
LIN {X 0,Y 559.161,Z 356.832,A -85,B 0,C 180,E1 -3028.981,E2 -3028.981} C_VEL
LIN {X 0,Y 559.164,Z 356.832,A -85,B 0,C 180,E1 -3031.617,E2 -3031.617} C_VEL
LIN {X 0,Y 559.192,Z 356.825,A -85,B 0,C 180,E1 -3033.903,E2 -3033.903} C_VEL
LIN {X 0,Y 559.156,Z 356.835,A -85,B 0,C 180,E1 -3037.068,E2 -3037.068} C_VEL
LIN {X 0,Y 559.181,Z 356.832,A -85,B 0,C 180,E1 -3039.395,E2 -3039.395} C_VEL
LIN {X 0,Y 559.157,Z 356.829,A -85,B 0,C 180,E1 -3042.443,E2 -3042.443} C_VEL
LIN {X 0,Y 559.186,Z 356.83,A -85,B 0,C 180,E1 -3045.442,E2 -3045.442} C_VEL
LIN {X 0,Y 559.216,Z 356.823,A -85,B 0,C 180,E1 -3048.593,E2 -3048.593} C_VEL
LIN {X 0,Y 559.196,Z 356.829,A -85,B 0,C 180,E1 -3051.326,E2 -3051.326} C_VEL
LIN {X 0,Y 559.224,Z 356.82,A -85,B 0,C 180,E1 -3054.23,E2 -3054.23} C_VEL
LIN {X 0,Y 559.24,Z 356.826,A -85,B 0,C 180,E1 -3057.119,E2 -3057.119} C_VEL
LIN {X 0,Y 559.252,Z 356.816,A -85,B 0,C 180,E1 -3060,E2 -3060} C_VEL
LIN {X 0,Y 559.24,Z 356.828,A -85,B 0,C 180,E1 -3062.881,E2 -3062.881} C_VEL
LIN {X 0,Y 559.223,Z 356.82,A -85,B 0,C 180,E1 -3065.77,E2 -3065.77} C_VEL
LIN {X 0,Y 559.196,Z 356.831,A -85,B 0,C 180,E1 -3068.674,E2 -3068.674} C_VEL
LIN {X 0,Y 559.2,Z 356.823,A -85,B 0,C 180,E1 -3071.601,E2 -3071.601} C_VEL
LIN {X 0,Y 559.19,Z 356.832,A -85,B 0,C 180,E1 -3074.596,E2 -3074.596} C_VEL
LIN {X 0,Y 559.157,Z 356.828,A -85,B 0,C 180,E1 -3077.557,E2 -3077.557} C_VEL
LIN {X 0,Y 559.167,Z 356.827,A -85,B 0,C 180,E1 -3079.838,E2 -3079.838} C_VEL
LIN {X 0,Y 559.148,Z 356.832,A -85,B 0,C 180,E1 -3082.153,E2 -3082.153} C_VEL
LIN {X 0,Y 559.153,Z 356.837,A -85,B 0,C 180,E1 -3084.505,E2 -3084.505} C_VEL
LIN {X 0,Y 559.172,Z 356.831,A -85,B 0,C 180,E1 -3086.902,E2 -3086.902} C_VEL
LIN {X 0,Y 559.143,Z 356.831,A -85,B 0,C 180,E1 -3089.859,E2 -3089.859} C_VEL
LIN {X 0,Y 559.139,Z 356.832,A -85,B 0,C 180,E1 -3090.637,E2 -3090.637} C_VEL
LIN {X 0,Y 558.481,Z 356.915,A -85,B 0,C 180,E1 -3091.239,E2 -3091.239} C_VEL
LIN {X 0,Y 555.619,Z 357.274,A -85,B 0,C 180,E1 -3092.215,E2 -3092.215} C_VEL
LIN {X 0,Y 553.204,Z 357.572,A -85,B 0,C 180,E1 -3093.001,E2 -3093.001} C_VEL
LIN {X 0,Y 552.182,Z 357.697,A -85,B 0,C 180,E1 -3093.607,E2 -3093.607} C_VEL
LIN {X 0,Y 552.108,Z 357.708,A -85,B 0,C 180,E1 -3093.813,E2 -3093.813} C_VEL
LIN {X 0,Y 552.109,Z 357.711,A -85,B 0,C 180,E1 -3096.747,E2 -3096.747} C_VEL
LIN {X 0,Y 552.129,Z 357.704,A -85,B 0,C 180,E1 -3099.528,E2 -3099.528} C_VEL
LIN {X 0,Y 552.127,Z 357.713,A -85,B 0,C 180,E1 -3102.426,E2 -3102.426} C_VEL
LIN {X 0,Y 552.094,Z 357.709,A -85,B 0,C 180,E1 -3105.564,E2 -3105.564} C_VEL
LIN {X 0,Y 552.129,Z 357.707,A -85,B 0,C 180,E1 -3108.678,E2 -3108.678} C_VEL
LIN {X 0,Y 552.118,Z 357.705,A -85,B 0,C 180,E1 -3111.412,E2 -3111.412} C_VEL
LIN {X 0,Y 552.113,Z 357.715,A -85,B 0,C 180,E1 -3114.159,E2 -3114.159} C_VEL
LIN {X 0,Y 552.115,Z 357.707,A -85,B 0,C 180,E1 -3116.815,E2 -3116.815} C_VEL
LIN {X 0,Y 552.129,Z 357.711,A -85,B 0,C 180,E1 -3119.948,E2 -3119.948} C_VEL
LIN {X 0,Y 552.14,Z 357.702,A -85,B 0,C 180,E1 -3123,E2 -3123} C_VEL
LIN {X 0,Y 552.114,Z 357.707,A -85,B 0,C 180,E1 -3125.162,E2 -3125.162} C_VEL
LIN {X 0,Y 552.128,Z 357.711,A -85,B 0,C 180,E1 -3128.338,E2 -3128.338} C_VEL
LIN {X 0,Y 552.163,Z 357.813,A -85,B 0,C 180,E1 -3130.624,E2 -3130.624} C_VEL
LIN {X 0,Y 552.527,Z 364.053,A -85,B 0,C 180,E1 -3131.843,E2 -3131.843} C_VEL
LIN {X 0,Y 552.257,Z 381.055,A -85,B 0,C 180,E1 -3135.067,E2 -3135.067} C_VEL
LIN {X 0,Y 552.218,Z 384.481,A -85,B 0,C 180,E1 -3135.693,E2 -3135.693} C_VEL
LIN {X 0,Y 553.427,Z 392.163,A -85,B 0,C 180,E1 -3135.826,E2 -3135.826} C_VEL
LIN {X 0,Y 553.123,Z 491.041,A -85,B 0,C 180,E1 -3137.13,E2 -3137.13} C_VEL
LIN {X 0,Y 552.999,Z 504.271,A -85,B 0,C 180,E1 -3137.453,E2 -3137.453} C_VEL
LIN {X 0,Y 552.847,Z 516.416,A -85,B 0,C 180,E1 -3137.893,E2 -3137.893} C_VEL
LIN {X 0,Y 552.693,Z 527.856,A -85,B 0,C 180,E1 -3138.448,E2 -3138.448} C_VEL
LIN {X 0,Y 552.491,Z 539.573,A -85,B 0,C 180,E1 -3139.186,E2 -3139.186} C_VEL
LIN {X 0,Y 552.304,Z 550.088,A -85,B 0,C 180,E1 -3140.016,E2 -3140.016} C_VEL
LIN {X 0,Y 552.153,Z 558.683,A -85,B 0,C 180,E1 -3140.845,E2 -3140.845} C_VEL
LIN {X 0,Y 552.007,Z 566.601,A -85,B 0,C 180,E1 -3141.765,E2 -3141.765} C_VEL
LIN {X 0,Y 551.895,Z 574.461,A -85,B 0,C 180,E1 -3142.886,E2 -3142.886} C_VEL
LIN {X 0,Y 551.868,Z 581.458,A -85,B 0,C 180,E1 -3144.153,E2 -3144.153} C_VEL
LIN {X 0,Y 551.725,Z 586.198,A -85,B 0,C 180,E1 -3145.251,E2 -3145.251} C_VEL
LIN {X 0,Y 551.75,Z 589.83,A -85,B 0,C 180,E1 -3146.349,E2 -3146.349} C_VEL
LIN {X 0,Y 551.723,Z 591.706,A -85,B 0,C 180,E1 -3147.079,E2 -3147.079} C_VEL
LIN {X 0,Y 551.657,Z 593.128,A -85,B 0,C 180,E1 -3147.81,E2 -3147.81} C_VEL
LIN {X 0,Y 551.642,Z 594.757,A -85,B 0,C 180,E1 -3149.27,E2 -3149.27} C_VEL
LIN {X 0,Y 551.641,Z 594.996,A -85,B 0,C 180,E1 -3150,E2 -3150} C_VEL
LIN {X 0,Y 551.641,Z 594.815,A -85,B 0,C 180,E1 -3150.73,E2 -3150.73} C_VEL
LIN {X 0,Y 551.657,Z 593.264,A -85,B 0,C 180,E1 -3152.19,E2 -3152.19} C_VEL
LIN {X 0,Y 551.724,Z 591.903,A -85,B 0,C 180,E1 -3152.921,E2 -3152.921} C_VEL
LIN {X 0,Y 551.764,Z 589.026,A -85,B 0,C 180,E1 -3154.017,E2 -3154.017} C_VEL
LIN {X 0,Y 551.724,Z 585.125,A -85,B 0,C 180,E1 -3155.116,E2 -3155.116} C_VEL
LIN {X 0,Y 551.811,Z 579.394,A -85,B 0,C 180,E1 -3156.349,E2 -3156.349} C_VEL
LIN {X 0,Y 551.925,Z 572.538,A -85,B 0,C 180,E1 -3157.499,E2 -3157.499} C_VEL
LIN {X 0,Y 552.063,Z 564.356,A -85,B 0,C 180,E1 -3158.603,E2 -3158.603} C_VEL
LIN {X 0,Y 552.197,Z 555.988,A -85,B 0,C 180,E1 -3159.523,E2 -3159.523} C_VEL
LIN {X 0,Y 552.406,Z 545.666,A -85,B 0,C 180,E1 -3160.445,E2 -3160.445} C_VEL
LIN {X 0,Y 552.608,Z 535.001,A -85,B 0,C 180,E1 -3161.212,E2 -3161.212} C_VEL
LIN {X 0,Y 552.747,Z 524.266,A -85,B 0,C 180,E1 -3161.831,E2 -3161.831} C_VEL
LIN {X 0,Y 552.907,Z 511.737,A -85,B 0,C 180,E1 -3162.386,E2 -3162.386} C_VEL
LIN {X 0,Y 553.041,Z 498.298,A -85,B 0,C 180,E1 -3162.802,E2 -3162.802} C_VEL
LIN {X 0,Y 553.153,Z 484.985,A -85,B 0,C 180,E1 -3163.056,E2 -3163.056} C_VEL
LIN {X 0,Y 553.398,Z 391.476,A -85,B 0,C 180,E1 -3164.274,E2 -3164.274} C_VEL
LIN {X 0,Y 552.193,Z 384.315,A -85,B 0,C 180,E1 -3164.419,E2 -3164.419} C_VEL
LIN {X 0,Y 552.406,Z 368.459,A -85,B 0,C 180,E1 -3167.409,E2 -3167.409} C_VEL
LIN {X 0,Y 552.488,Z 360.536,A -85,B 0,C 180,E1 -3168.927,E2 -3168.927} C_VEL
LIN {X 0,Y 552.153,Z 357.709,A -85,B 0,C 180,E1 -3169.534,E2 -3169.534} C_VEL
LIN {X 0,Y 552.098,Z 357.715,A -85,B 0,C 180,E1 -3172.45,E2 -3172.45} C_VEL
LIN {X 0,Y 552.157,Z 357.704,A -85,B 0,C 180,E1 -3175.35,E2 -3175.35} C_VEL
LIN {X 0,Y 552.121,Z 357.713,A -85,B 0,C 180,E1 -3178.097,E2 -3178.097} C_VEL
LIN {X 0,Y 552.107,Z 357.708,A -85,B 0,C 180,E1 -3180.608,E2 -3180.608} C_VEL
LIN {X 0,Y 552.123,Z 357.705,A -85,B 0,C 180,E1 -3183.184,E2 -3183.184} C_VEL
LIN {X 0,Y 552.113,Z 357.715,A -85,B 0,C 180,E1 -3185.841,E2 -3185.841} C_VEL
LIN {X 0,Y 552.123,Z 357.705,A -85,B 0,C 180,E1 -3189.061,E2 -3189.061} C_VEL
LIN {X 0,Y 552.125,Z 357.709,A -85,B 0,C 180,E1 -3191.444,E2 -3191.444} C_VEL
LIN {X 0,Y 552.091,Z 357.709,A -85,B 0,C 180,E1 -3194.531,E2 -3194.531} C_VEL
LIN {X 0,Y 552.127,Z 357.712,A -85,B 0,C 180,E1 -3197.584,E2 -3197.584} C_VEL
LIN {X 0,Y 552.129,Z 357.704,A -85,B 0,C 180,E1 -3200.472,E2 -3200.472} C_VEL
LIN {X 0,Y 552.116,Z 357.71,A -85,B 0,C 180,E1 -3203.314,E2 -3203.314} C_VEL
LIN {X 0,Y 552.133,Z 357.708,A -85,B 0,C 180,E1 -3205.939,E2 -3205.939} C_VEL
LIN {X 0,Y 552.112,Z 357.706,A -85,B 0,C 180,E1 -3208.54,E2 -3208.54} C_VEL
LIN {X 0,Y 552.119,Z 357.714,A -85,B 0,C 180,E1 -3211.437,E2 -3211.437} C_VEL
LIN {X 0,Y 552.129,Z 357.704,A -85,B 0,C 180,E1 -3214.356,E2 -3214.356} C_VEL
LIN {X 0,Y 552.132,Z 357.704,A -85,B 0,C 180,E1 -3216.759,E2 -3216.759} C_VEL
LIN {X 0,Y 552.12,Z 357.71,A -85,B 0,C 180,E1 -3219.12,E2 -3219.12} C_VEL
LIN {X 0,Y 552.125,Z 357.713,A -85,B 0,C 180,E1 -3221.444,E2 -3221.444} C_VEL
LIN {X 0,Y 552.115,Z 357.709,A -85,B 0,C 180,E1 -3223.737,E2 -3223.737} C_VEL
LIN {X 0,Y 552.129,Z 357.705,A -85,B 0,C 180,E1 -3226.004,E2 -3226.004} C_VEL
LIN {X 0,Y 552.17,Z 357.704,A -85,B 0,C 180,E1 -3228.993,E2 -3228.993} C_VEL
LIN {X 0,Y 552.158,Z 357.701,A -85,B 0,C 180,E1 -3231.951,E2 -3231.951} C_VEL
LIN {X 0,Y 552.227,Z 357.697,A -85,B 0,C 180,E1 -3234.889,E2 -3234.889} C_VEL
LIN {X 0,Y 552.216,Z 357.694,A -85,B 0,C 180,E1 -3237.812,E2 -3237.812} C_VEL
LIN {X 0,Y 552.24,Z 357.694,A -85,B 0,C 180,E1 -3240.729,E2 -3240.729} C_VEL
LIN {X 0,Y 552.205,Z 357.702,A -85,B 0,C 180,E1 -3242.918,E2 -3242.918} C_VEL
LIN {X 0,Y 552.194,Z 357.696,A -85,B 0,C 180,E1 -3245.844,E2 -3245.844} C_VEL
LIN {X 0,Y 552.164,Z 357.706,A -85,B 0,C 180,E1 -3248.786,E2 -3248.786} C_VEL
LIN {X 0,Y 552.156,Z 357.701,A -85,B 0,C 180,E1 -3251.751,E2 -3251.751} C_VEL
LIN {X 0,Y 552.128,Z 357.711,A -85,B 0,C 180,E1 -3254.749,E2 -3254.749} C_VEL
LIN {X 0,Y 552.108,Z 357.706,A -85,B 0,C 180,E1 -3257.789,E2 -3257.789} C_VEL
LIN {X 0,Y 552.128,Z 357.705,A -85,B 0,C 180,E1 -3260.101,E2 -3260.101} C_VEL
LIN {X 0,Y 552.107,Z 357.711,A -85,B 0,C 180,E1 -3262.45,E2 -3262.45} C_VEL
LIN {X 0,Y 552.149,Z 357.703,A -85,B 0,C 180,E1 -3265.351,E2 -3265.351} C_VEL
LIN {X 0,Y 552.121,Z 357.706,A -85,B 0,C 180,E1 -3268.098,E2 -3268.098} C_VEL
LIN {X 0,Y 552.101,Z 357.716,A -85,B 0,C 180,E1 -3270.609,E2 -3270.609} C_VEL
LIN {X 0,Y 552.123,Z 357.707,A -85,B 0,C 180,E1 -3273.185,E2 -3273.185} C_VEL
LIN {X 0,Y 552.108,Z 357.707,A -85,B 0,C 180,E1 -3275.842,E2 -3275.842} C_VEL
LIN {X 0,Y 552.121,Z 357.707,A -85,B 0,C 180,E1 -3279.063,E2 -3279.063} C_VEL
LIN {X 0,Y 552.136,Z 357.703,A -85,B 0,C 180,E1 -3281.445,E2 -3281.445} C_VEL
LIN {X 0,Y 552.093,Z 357.717,A -85,B 0,C 180,E1 -3284.533,E2 -3284.533} C_VEL
LIN {X 0,Y 552.127,Z 357.704,A -85,B 0,C 180,E1 -3287.585,E2 -3287.585} C_VEL
LIN {X 0,Y 552.132,Z 357.712,A -85,B 0,C 180,E1 -3290.474,E2 -3290.474} C_VEL
LIN {X 0,Y 552.113,Z 357.706,A -85,B 0,C 180,E1 -3293.316,E2 -3293.316} C_VEL
LIN {X 0,Y 552.131,Z 357.708,A -85,B 0,C 180,E1 -3295.94,E2 -3295.94} C_VEL
LIN {X 0,Y 552.118,Z 357.711,A -85,B 0,C 180,E1 -3298.541,E2 -3298.541} C_VEL
LIN {X 0,Y 552.124,Z 357.706,A -85,B 0,C 180,E1 -3301.439,E2 -3301.439} C_VEL
LIN {X 0,Y 552.131,Z 357.713,A -85,B 0,C 180,E1 -3304.356,E2 -3304.356} C_VEL
LIN {X 0,Y 552.172,Z 357.903,A -85,B 0,C 180,E1 -3306.053,E2 -3306.053} C_VEL
LIN {X 0,Y 553.217,Z 363.941,A -85,B 0,C 180,E1 -3307.006,E2 -3307.006} C_VEL
LIN {X 0,Y 552.967,Z 382.32,A -85,B 0,C 180,E1 -3309.737,E2 -3309.737} C_VEL
LIN {X 0,Y 552.657,Z 402.932,A -85,B 0,C 180,E1 -3312.75,E2 -3312.75} C_VEL
LIN {X 0,Y 552.382,Z 422.702,A -85,B 0,C 180,E1 -3315.624,E2 -3315.624} C_VEL
LIN {X 0,Y 553.451,Z 430.711,A -85,B 0,C 180,E1 -3315.763,E2 -3315.763} C_VEL
LIN {X 0,Y 553.113,Z 530.961,A -85,B 0,C 180,E1 -3317.083,E2 -3317.083} C_VEL
LIN {X 0,Y 553.008,Z 544.227,A -85,B 0,C 180,E1 -3317.407,E2 -3317.407} C_VEL
LIN {X 0,Y 552.846,Z 556.377,A -85,B 0,C 180,E1 -3317.846,E2 -3317.846} C_VEL
LIN {X 0,Y 552.647,Z 567.256,A -85,B 0,C 180,E1 -3318.37,E2 -3318.37} C_VEL
LIN {X 0,Y 552.52,Z 578.908,A -85,B 0,C 180,E1 -3319.094,E2 -3319.094} C_VEL
LIN {X 0,Y 552.294,Z 589.54,A -85,B 0,C 180,E1 -3319.923,E2 -3319.923} C_VEL
LIN {X 0,Y 552.125,Z 599.115,A -85,B 0,C 180,E1 -3320.845,E2 -3320.845} C_VEL
LIN {X 0,Y 552.013,Z 606.962,A -85,B 0,C 180,E1 -3321.765,E2 -3321.765} C_VEL
LIN {X 0,Y 551.889,Z 614.623,A -85,B 0,C 180,E1 -3322.868,E2 -3322.868} C_VEL
LIN {X 0,Y 551.867,Z 621.68,A -85,B 0,C 180,E1 -3324.153,E2 -3324.153} C_VEL
LIN {X 0,Y 551.725,Z 626.373,A -85,B 0,C 180,E1 -3325.251,E2 -3325.251} C_VEL
LIN {X 0,Y 551.75,Z 629.958,A -85,B 0,C 180,E1 -3326.349,E2 -3326.349} C_VEL
LIN {X 0,Y 551.723,Z 631.807,A -85,B 0,C 180,E1 -3327.079,E2 -3327.079} C_VEL
LIN {X 0,Y 551.645,Z 634.184,A -85,B 0,C 180,E1 -3328.54,E2 -3328.54} C_VEL
LIN {X 0,Y 551.64,Z 635,A -85,B 0,C 180,E1 -3330,E2 -3330} C_VEL
LIN {X 0,Y 551.645,Z 634.185,A -85,B 0,C 180,E1 -3331.46,E2 -3331.46} C_VEL
LIN {X 0,Y 551.723,Z 631.81,A -85,B 0,C 180,E1 -3332.921,E2 -3332.921} C_VEL
LIN {X 0,Y 551.763,Z 628.896,A -85,B 0,C 180,E1 -3334.017,E2 -3334.017} C_VEL
LIN {X 0,Y 551.724,Z 624.949,A -85,B 0,C 180,E1 -3335.116,E2 -3335.116} C_VEL
LIN {X 0,Y 551.815,Z 619.124,A -85,B 0,C 180,E1 -3336.353,E2 -3336.353} C_VEL
LIN {X 0,Y 551.926,Z 612.237,A -85,B 0,C 180,E1 -3337.499,E2 -3337.499} C_VEL
LIN {X 0,Y 552.082,Z 603.993,A -85,B 0,C 180,E1 -3338.602,E2 -3338.602} C_VEL
LIN {X 0,Y 552.221,Z 595.542,A -85,B 0,C 180,E1 -3339.523,E2 -3339.523} C_VEL
LIN {X 0,Y 552.432,Z 585.096,A -85,B 0,C 180,E1 -3340.445,E2 -3340.445} C_VEL
LIN {X 0,Y 552.555,Z 574.291,A -85,B 0,C 180,E1 -3341.214,E2 -3341.214} C_VEL
LIN {X 0,Y 552.781,Z 563.411,A -85,B 0,C 180,E1 -3341.83,E2 -3341.83} C_VEL
LIN {X 0,Y 552.884,Z 551.772,A -85,B 0,C 180,E1 -3342.34,E2 -3342.34} C_VEL
LIN {X 0,Y 553.057,Z 538.357,A -85,B 0,C 180,E1 -3342.755,E2 -3342.755} C_VEL
LIN {X 0,Y 553.175,Z 525.105,A -85,B 0,C 180,E1 -3343.009,E2 -3343.009} C_VEL
LIN {X 0,Y 553.414,Z 429.543,A -85,B 0,C 180,E1 -3344.254,E2 -3344.254} C_VEL
LIN {X 0,Y 552.39,Z 422.651,A -85,B 0,C 180,E1 -3344.383,E2 -3344.383} C_VEL
LIN {X 0,Y 552.684,Z 401.205,A -85,B 0,C 180,E1 -3347.501,E2 -3347.501} C_VEL
LIN {X 0,Y 552.964,Z 381.006,A -85,B 0,C 180,E1 -3350.457,E2 -3350.457} C_VEL
LIN {X 0,Y 553.216,Z 363.929,A -85,B 0,C 180,E1 -3352.994,E2 -3352.994} C_VEL
LIN {X 0,Y 552.145,Z 357.712,A -85,B 0,C 180,E1 -3353.978,E2 -3353.978} C_VEL
LIN {X 0,Y 552.121,Z 357.707,A -85,B 0,C 180,E1 -3356.456,E2 -3356.456} C_VEL
LIN {X 0,Y 552.11,Z 357.708,A -85,B 0,C 180,E1 -3358.928,E2 -3358.928} C_VEL
LIN {X 0,Y 552.135,Z 357.71,A -85,B 0,C 180,E1 -3361.479,E2 -3361.479} C_VEL
LIN {X 0,Y 552.138,Z 357.706,A -85,B 0,C 180,E1 -3364.171,E2 -3364.171} C_VEL
LIN {X 0,Y 552.11,Z 357.706,A -85,B 0,C 180,E1 -3366.746,E2 -3366.746} C_VEL
LIN {X 0,Y 552.132,Z 357.712,A -85,B 0,C 180,E1 -3369.526,E2 -3369.526} C_VEL
LIN {X 0,Y 552.127,Z 357.704,A -85,B 0,C 180,E1 -3372.425,E2 -3372.425} C_VEL
LIN {X 0,Y 552.096,Z 357.718,A -85,B 0,C 180,E1 -3375.562,E2 -3375.562} C_VEL
LIN {X 0,Y 552.136,Z 357.703,A -85,B 0,C 180,E1 -3378.675,E2 -3378.675} C_VEL
LIN {X 0,Y 552.115,Z 357.715,A -85,B 0,C 180,E1 -3381.411,E2 -3381.411} C_VEL
LIN {X 0,Y 552.107,Z 357.707,A -85,B 0,C 180,E1 -3384.158,E2 -3384.158} C_VEL
LIN {X 0,Y 552.123,Z 357.706,A -85,B 0,C 180,E1 -3386.815,E2 -3386.815} C_VEL
LIN {X 0,Y 552.108,Z 357.716,A -85,B 0,C 180,E1 -3389.391,E2 -3389.391} C_VEL
LIN {X 0,Y 552.12,Z 357.707,A -85,B 0,C 180,E1 -3391.902,E2 -3391.902} C_VEL
LIN {X 0,Y 552.149,Z 357.703,A -85,B 0,C 180,E1 -3394.649,E2 -3394.649} C_VEL
LIN {X 0,Y 552.107,Z 357.711,A -85,B 0,C 180,E1 -3397.55,E2 -3397.55} C_VEL
LIN {X 0,Y 552.149,Z 357.703,A -85,B 0,C 180,E1 -3400.674,E2 -3400.674} C_VEL
LIN {X 0,Y 552.115,Z 357.707,A -85,B 0,C 180,E1 -3403.737,E2 -3403.737} C_VEL
LIN {X 0,Y 552.129,Z 357.704,A -85,B 0,C 180,E1 -3406.004,E2 -3406.004} C_VEL
LIN {X 0,Y 552.185,Z 357.705,A -85,B 0,C 180,E1 -3408.994,E2 -3408.994} C_VEL
LIN {X 0,Y 552.158,Z 357.7,A -85,B 0,C 180,E1 -3411.952,E2 -3411.952} C_VEL
LIN {X 0,Y 552.227,Z 357.699,A -85,B 0,C 180,E1 -3414.889,E2 -3414.889} C_VEL
LIN {X 0,Y 552.216,Z 357.693,A -85,B 0,C 180,E1 -3417.812,E2 -3417.812} C_VEL
LIN {X 0,Y 552.241,Z 357.696,A -85,B 0,C 180,E1 -3420.729,E2 -3420.729} C_VEL
LIN {X 0,Y 552.205,Z 357.704,A -85,B 0,C 180,E1 -3422.918,E2 -3422.918} C_VEL
LIN {X 0,Y 552.193,Z 357.696,A -85,B 0,C 180,E1 -3425.844,E2 -3425.844} C_VEL
LIN {X 0,Y 552.164,Z 357.709,A -85,B 0,C 180,E1 -3428.786,E2 -3428.786} C_VEL
LIN {X 0,Y 552.156,Z 357.7,A -85,B 0,C 180,E1 -3431.751,E2 -3431.751} C_VEL
LIN {X 0,Y 552.128,Z 357.714,A -85,B 0,C 180,E1 -3434.749,E2 -3434.749} C_VEL
LIN {X 0,Y 552.108,Z 357.706,A -85,B 0,C 180,E1 -3437.789,E2 -3437.789} C_VEL
LIN {X 0,Y 552.127,Z 357.706,A -85,B 0,C 180,E1 -3440.101,E2 -3440.101} C_VEL
LIN {X 0,Y 552.107,Z 357.713,A -85,B 0,C 180,E1 -3442.45,E2 -3442.45} C_VEL
LIN {X 0,Y 552.149,Z 357.702,A -85,B 0,C 180,E1 -3445.351,E2 -3445.351} C_VEL
LIN {X 0,Y 552.12,Z 357.708,A -85,B 0,C 180,E1 -3448.098,E2 -3448.098} C_VEL
LIN {X 0,Y 552.1,Z 357.715,A -85,B 0,C 180,E1 -3450.633,E2 -3450.633} C_VEL
LIN {X 0,Y 552.117,Z 357.706,A -85,B 0,C 180,E1 -3453.186,E2 -3453.186} C_VEL
LIN {X 0,Y 552.108,Z 357.708,A -85,B 0,C 180,E1 -3453.813,E2 -3453.813} C_VEL
LIN {X 0,Y 551.472,Z 357.795,A -85,B 0,C 180,E1 -3454.421,E2 -3454.421} C_VEL
LIN {X 0,Y 548.651,Z 358.145,A -85,B 0,C 180,E1 -3455.41,E2 -3455.41} C_VEL
LIN {X 0,Y 546.231,Z 358.445,A -85,B 0,C 180,E1 -3456.205,E2 -3456.205} C_VEL
LIN {X 0,Y 545.162,Z 358.576,A -85,B 0,C 180,E1 -3456.819,E2 -3456.819} C_VEL
LIN {X 0,Y 545.06,Z 358.586,A -85,B 0,C 180,E1 -3457.027,E2 -3457.027} C_VEL
LIN {X 0,Y 545.087,Z 358.587,A -85,B 0,C 180,E1 -3460.141,E2 -3460.141} C_VEL
LIN {X 0,Y 545.084,Z 358.582,A -85,B 0,C 180,E1 -3463.106,E2 -3463.106} C_VEL
LIN {X 0,Y 545.053,Z 358.594,A -85,B 0,C 180,E1 -3466.226,E2 -3466.226} C_VEL
LIN {X 0,Y 545.088,Z 358.582,A -85,B 0,C 180,E1 -3468.887,E2 -3468.887} C_VEL
LIN {X 0,Y 545.052,Z 358.588,A -85,B 0,C 180,E1 -3471.764,E2 -3471.764} C_VEL
LIN {X 0,Y 545.065,Z 358.588,A -85,B 0,C 180,E1 -3474.535,E2 -3474.535} C_VEL
LIN {X 0,Y 545.069,Z 358.583,A -85,B 0,C 180,E1 -3477.212,E2 -3477.212} C_VEL
LIN {X 0,Y 545.085,Z 358.586,A -85,B 0,C 180,E1 -3479.813,E2 -3479.813} C_VEL
LIN {X 0,Y 545.094,Z 358.581,A -85,B 0,C 180,E1 -3482.827,E2 -3482.827} C_VEL
LIN {X 0,Y 545.05,Z 358.591,A -85,B 0,C 180,E1 -3485.631,E2 -3485.631} C_VEL
LIN {X 0,Y 545.066,Z 358.587,A -85,B 0,C 180,E1 -3488.837,E2 -3488.837} C_VEL
LIN {X 0,Y 545.17,Z 358.774,A -85,B 0,C 180,E1 -3490.515,E2 -3490.515} C_VEL
LIN {X 0,Y 545.56,Z 365.272,A -85,B 0,C 180,E1 -3491.797,E2 -3491.797} C_VEL
LIN {X 0,Y 545.244,Z 382.291,A -85,B 0,C 180,E1 -3495.061,E2 -3495.061} C_VEL
LIN {X 0,Y 545.18,Z 384.605,A -85,B 0,C 180,E1 -3495.502,E2 -3495.502} C_VEL
LIN {X 0,Y 546.559,Z 392.815,A -85,B 0,C 180,E1 -3495.65,E2 -3495.65} C_VEL
LIN {X 0,Y 546.216,Z 491.106,A -85,B 0,C 180,E1 -3496.964,E2 -3496.964} C_VEL
LIN {X 0,Y 546.075,Z 504.306,A -85,B 0,C 180,E1 -3497.291,E2 -3497.291} C_VEL
LIN {X 0,Y 545.895,Z 516.419,A -85,B 0,C 180,E1 -3497.736,E2 -3497.736} C_VEL
LIN {X 0,Y 545.728,Z 528.613,A -85,B 0,C 180,E1 -3498.342,E2 -3498.342} C_VEL
LIN {X 0,Y 545.503,Z 539.579,A -85,B 0,C 180,E1 -3499.046,E2 -3499.046} C_VEL
LIN {X 0,Y 545.268,Z 550.094,A -85,B 0,C 180,E1 -3499.886,E2 -3499.886} C_VEL
LIN {X 0,Y 545.122,Z 558.688,A -85,B 0,C 180,E1 -3500.726,E2 -3500.726} C_VEL
LIN {X 0,Y 544.975,Z 566.606,A -85,B 0,C 180,E1 -3501.658,E2 -3501.658} C_VEL
LIN {X 0,Y 544.829,Z 574.353,A -85,B 0,C 180,E1 -3502.775,E2 -3502.775} C_VEL
LIN {X 0,Y 544.778,Z 581.46,A -85,B 0,C 180,E1 -3504.076,E2 -3504.076} C_VEL
LIN {X 0,Y 544.629,Z 586.2,A -85,B 0,C 180,E1 -3505.189,E2 -3505.189} C_VEL
LIN {X 0,Y 544.669,Z 589.831,A -85,B 0,C 180,E1 -3506.301,E2 -3506.301} C_VEL
LIN {X 0,Y 544.65,Z 591.708,A -85,B 0,C 180,E1 -3507.041,E2 -3507.041} C_VEL
LIN {X 0,Y 544.571,Z 593.128,A -85,B 0,C 180,E1 -3507.781,E2 -3507.781} C_VEL
LIN {X 0,Y 544.542,Z 594.757,A -85,B 0,C 180,E1 -3509.261,E2 -3509.261} C_VEL
LIN {X 0,Y 544.542,Z 594.996,A -85,B 0,C 180,E1 -3510,E2 -3510} C_VEL
LIN {X 0,Y 544.542,Z 594.815,A -85,B 0,C 180,E1 -3510.739,E2 -3510.739} C_VEL
LIN {X 0,Y 544.572,Z 593.262,A -85,B 0,C 180,E1 -3512.219,E2 -3512.219} C_VEL
LIN {X 0,Y 544.651,Z 591.901,A -85,B 0,C 180,E1 -3512.959,E2 -3512.959} C_VEL
LIN {X 0,Y 544.684,Z 589.024,A -85,B 0,C 180,E1 -3514.069,E2 -3514.069} C_VEL
LIN {X 0,Y 544.653,Z 585.123,A -85,B 0,C 180,E1 -3515.182,E2 -3515.182} C_VEL
LIN {X 0,Y 544.724,Z 579.898,A -85,B 0,C 180,E1 -3516.335,E2 -3516.335} C_VEL
LIN {X 0,Y 544.859,Z 572.533,A -85,B 0,C 180,E1 -3517.597,E2 -3517.597} C_VEL
LIN {X 0,Y 544.999,Z 564.351,A -85,B 0,C 180,E1 -3518.715,E2 -3518.715} C_VEL
LIN {X 0,Y 545.158,Z 555.982,A -85,B 0,C 180,E1 -3519.648,E2 -3519.648} C_VEL
LIN {X 0,Y 545.382,Z 545.657,A -85,B 0,C 180,E1 -3520.581,E2 -3520.581} C_VEL
LIN {X 0,Y 545.672,Z 534.276,A -85,B 0,C 180,E1 -3521.403,E2 -3521.403} C_VEL
LIN {X 0,Y 545.81,Z 524.253,A -85,B 0,C 180,E1 -3521.983,E2 -3521.983} C_VEL
LIN {X 0,Y 545.964,Z 511.724,A -85,B 0,C 180,E1 -3522.546,E2 -3522.546} C_VEL
LIN {X 0,Y 546.128,Z 498.302,A -85,B 0,C 180,E1 -3522.967,E2 -3522.967} C_VEL
LIN {X 0,Y 546.254,Z 484.985,A -85,B 0,C 180,E1 -3523.224,E2 -3523.224} C_VEL
LIN {X 0,Y 546.488,Z 392.034,A -85,B 0,C 180,E1 -3524.452,E2 -3524.452} C_VEL
LIN {X 0,Y 545.176,Z 384.534,A -85,B 0,C 180,E1 -3524.603,E2 -3524.603} C_VEL
LIN {X 0,Y 545.45,Z 369.154,A -85,B 0,C 180,E1 -3527.546,E2 -3527.546} C_VEL
LIN {X 0,Y 545.43,Z 360.731,A -85,B 0,C 180,E1 -3529.182,E2 -3529.182} C_VEL
LIN {X 0,Y 545.105,Z 358.588,A -85,B 0,C 180,E1 -3529.655,E2 -3529.655} C_VEL
LIN {X 0,Y 545.047,Z 358.591,A -85,B 0,C 180,E1 -3532.757,E2 -3532.757} C_VEL
LIN {X 0,Y 545.096,Z 358.585,A -85,B 0,C 180,E1 -3535.508,E2 -3535.508} C_VEL
LIN {X 0,Y 545.103,Z 358.581,A -85,B 0,C 180,E1 -3538.492,E2 -3538.492} C_VEL
LIN {X 0,Y 545.068,Z 358.584,A -85,B 0,C 180,E1 -3541.047,E2 -3541.047} C_VEL
LIN {X 0,Y 545.071,Z 358.589,A -85,B 0,C 180,E1 -3543.671,E2 -3543.671} C_VEL
LIN {X 0,Y 545.055,Z 358.587,A -85,B 0,C 180,E1 -3546.378,E2 -3546.378} C_VEL
LIN {X 0,Y 545.103,Z 358.581,A -85,B 0,C 180,E1 -3549.323,E2 -3549.323} C_VEL
LIN {X 0,Y 545.076,Z 358.587,A -85,B 0,C 180,E1 -3552.102,E2 -3552.102} C_VEL
LIN {X 0,Y 545.059,Z 358.586,A -85,B 0,C 180,E1 -3555.166,E2 -3555.166} C_VEL
LIN {X 0,Y 545.079,Z 358.589,A -85,B 0,C 180,E1 -3557.897,E2 -3557.897} C_VEL
LIN {X 0,Y 545.1,Z 358.579,A -85,B 0,C 180,E1 -3560.675,E2 -3560.675} C_VEL
LIN {X 0,Y 545.055,Z 358.595,A -85,B 0,C 180,E1 -3563.62,E2 -3563.62} C_VEL
LIN {X 0,Y 545.071,Z 358.584,A -85,B 0,C 180,E1 -3566.328,E2 -3566.328} C_VEL
LIN {X 0,Y 545.061,Z 358.586,A -85,B 0,C 180,E1 -3568.952,E2 -3568.952} C_VEL
LIN {X 0,Y 545.098,Z 358.59,A -85,B 0,C 180,E1 -3571.507,E2 -3571.507} C_VEL
LIN {X 0,Y 545.092,Z 358.58,A -85,B 0,C 180,E1 -3574.489,E2 -3574.489} C_VEL
LIN {X 0,Y 545.06,Z 358.591,A -85,B 0,C 180,E1 -3577.243,E2 -3577.243} C_VEL
LIN {X 0,Y 545.113,Z 358.578,A -85,B 0,C 180,E1 -3580.414,E2 -3580.414} C_VEL
LIN {X 0,Y 545.071,Z 358.59,A -85,B 0,C 180,E1 -3583.521,E2 -3583.521} C_VEL
LIN {X 0,Y 545.087,Z 358.583,A -85,B 0,C 180,E1 -3585.82,E2 -3585.82} C_VEL
LIN {X 0,Y 545.124,Z 358.58,A -85,B 0,C 180,E1 -3588.849,E2 -3588.849} C_VEL
LIN {X 0,Y 545.128,Z 358.577,A -85,B 0,C 180,E1 -3591.847,E2 -3591.847} C_VEL
LIN {X 0,Y 545.201,Z 358.571,A -85,B 0,C 180,E1 -3594.823,E2 -3594.823} C_VEL
LIN {X 0,Y 545.188,Z 358.57,A -85,B 0,C 180,E1 -3597.784,E2 -3597.784} C_VEL
LIN {X 0,Y 545.209,Z 358.57,A -85,B 0,C 180,E1 -3600.739,E2 -3600.739} C_VEL
LIN {X 0,Y 545.171,Z 358.579,A -85,B 0,C 180,E1 -3602.956,E2 -3602.956} C_VEL
LIN {X 0,Y 545.165,Z 358.571,A -85,B 0,C 180,E1 -3605.92,E2 -3605.92} C_VEL
LIN {X 0,Y 545.121,Z 358.585,A -85,B 0,C 180,E1 -3608.9,E2 -3608.9} C_VEL
LIN {X 0,Y 545.127,Z 358.576,A -85,B 0,C 180,E1 -3611.904,E2 -3611.904} C_VEL
LIN {X 0,Y 545.077,Z 358.591,A -85,B 0,C 180,E1 -3614.944,E2 -3614.944} C_VEL
LIN {X 0,Y 545.076,Z 358.583,A -85,B 0,C 180,E1 -3618.026,E2 -3618.026} C_VEL
LIN {X 0,Y 545.093,Z 358.583,A -85,B 0,C 180,E1 -3620.372,E2 -3620.372} C_VEL
LIN {X 0,Y 545.106,Z 358.579,A -85,B 0,C 180,E1 -3623.558,E2 -3623.558} C_VEL
LIN {X 0,Y 545.082,Z 358.582,A -85,B 0,C 180,E1 -3626.001,E2 -3626.001} C_VEL
LIN {X 0,Y 545.084,Z 358.59,A -85,B 0,C 180,E1 -3628.749,E2 -3628.749} C_VEL
LIN {X 0,Y 545.071,Z 358.583,A -85,B 0,C 180,E1 -3631.683,E2 -3631.683} C_VEL
LIN {X 0,Y 545.079,Z 358.591,A -85,B 0,C 180,E1 -3634.563,E2 -3634.563} C_VEL
LIN {X 0,Y 545.034,Z 358.588,A -85,B 0,C 180,E1 -3637.304,E2 -3637.304} C_VEL
LIN {X 0,Y 545.088,Z 358.585,A -85,B 0,C 180,E1 -3640.141,E2 -3640.141} C_VEL
LIN {X 0,Y 545.084,Z 358.583,A -85,B 0,C 180,E1 -3643.106,E2 -3643.106} C_VEL
LIN {X 0,Y 545.061,Z 358.59,A -85,B 0,C 180,E1 -3646.225,E2 -3646.225} C_VEL
LIN {X 0,Y 545.094,Z 358.583,A -85,B 0,C 180,E1 -3648.888,E2 -3648.888} C_VEL
LIN {X 0,Y 545.052,Z 358.587,A -85,B 0,C 180,E1 -3651.764,E2 -3651.764} C_VEL
LIN {X 0,Y 545.065,Z 358.59,A -85,B 0,C 180,E1 -3654.535,E2 -3654.535} C_VEL
LIN {X 0,Y 545.081,Z 358.582,A -85,B 0,C 180,E1 -3657.213,E2 -3657.213} C_VEL
LIN {X 0,Y 545.066,Z 358.587,A -85,B 0,C 180,E1 -3659.811,E2 -3659.811} C_VEL
LIN {X 0,Y 545.089,Z 358.589,A -85,B 0,C 180,E1 -3662.345,E2 -3662.345} C_VEL
LIN {X 0,Y 545.118,Z 358.583,A -85,B 0,C 180,E1 -3664.821,E2 -3664.821} C_VEL
LIN {X 0,Y 545.117,Z 358.67,A -85,B 0,C 180,E1 -3665.877,E2 -3665.877} C_VEL
LIN {X 0,Y 546.338,Z 366.337,A -85,B 0,C 180,E1 -3667.1,E2 -3667.1} C_VEL
LIN {X 0,Y 545.945,Z 386.45,A -85,B 0,C 180,E1 -3670.119,E2 -3670.119} C_VEL
LIN {X 0,Y 545.593,Z 406.985,A -85,B 0,C 180,E1 -3673.153,E2 -3673.153} C_VEL
LIN {X 0,Y 545.38,Z 422.634,A -85,B 0,C 180,E1 -3675.435,E2 -3675.435} C_VEL
LIN {X 0,Y 546.566,Z 431.581,A -85,B 0,C 180,E1 -3675.591,E2 -3675.591} C_VEL
LIN {X 0,Y 546.207,Z 530.961,A -85,B 0,C 180,E1 -3676.916,E2 -3676.916} C_VEL
LIN {X 0,Y 546.084,Z 544.226,A -85,B 0,C 180,E1 -3677.244,E2 -3677.244} C_VEL
LIN {X 0,Y 545.901,Z 556.375,A -85,B 0,C 180,E1 -3677.689,E2 -3677.689} C_VEL
LIN {X 0,Y 545.678,Z 567.469,A -85,B 0,C 180,E1 -3678.231,E2 -3678.231} C_VEL
LIN {X 0,Y 545.529,Z 578.906,A -85,B 0,C 180,E1 -3678.952,E2 -3678.952} C_VEL
LIN {X 0,Y 545.286,Z 589.539,A -85,B 0,C 180,E1 -3679.792,E2 -3679.792} C_VEL
LIN {X 0,Y 545.084,Z 599.115,A -85,B 0,C 180,E1 -3680.726,E2 -3680.726} C_VEL
LIN {X 0,Y 544.977,Z 606.962,A -85,B 0,C 180,E1 -3681.658,E2 -3681.658} C_VEL
LIN {X 0,Y 544.823,Z 614.622,A -85,B 0,C 180,E1 -3682.775,E2 -3682.775} C_VEL
LIN {X 0,Y 544.776,Z 621.68,A -85,B 0,C 180,E1 -3684.076,E2 -3684.076} C_VEL
LIN {X 0,Y 544.629,Z 626.373,A -85,B 0,C 180,E1 -3685.189,E2 -3685.189} C_VEL
LIN {X 0,Y 544.669,Z 629.958,A -85,B 0,C 180,E1 -3686.301,E2 -3686.301} C_VEL
LIN {X 0,Y 544.65,Z 631.807,A -85,B 0,C 180,E1 -3687.041,E2 -3687.041} C_VEL
LIN {X 0,Y 544.546,Z 634.183,A -85,B 0,C 180,E1 -3688.521,E2 -3688.521} C_VEL
LIN {X 0,Y 544.541,Z 635,A -85,B 0,C 180,E1 -3690,E2 -3690} C_VEL
LIN {X 0,Y 544.546,Z 634.184,A -85,B 0,C 180,E1 -3691.479,E2 -3691.479} C_VEL
LIN {X 0,Y 544.65,Z 631.81,A -85,B 0,C 180,E1 -3692.959,E2 -3692.959} C_VEL
LIN {X 0,Y 544.683,Z 628.896,A -85,B 0,C 180,E1 -3694.069,E2 -3694.069} C_VEL
LIN {X 0,Y 544.654,Z 624.949,A -85,B 0,C 180,E1 -3695.182,E2 -3695.182} C_VEL
LIN {X 0,Y 544.73,Z 619.643,A -85,B 0,C 180,E1 -3696.34,E2 -3696.34} C_VEL
LIN {X 0,Y 544.836,Z 613.468,A -85,B 0,C 180,E1 -3697.411,E2 -3697.411} C_VEL
LIN {X 0,Y 545.006,Z 605.479,A -85,B 0,C 180,E1 -3698.528,E2 -3698.528} C_VEL
LIN {X 0,Y 545.152,Z 597.335,A -85,B 0,C 180,E1 -3699.46,E2 -3699.46} C_VEL
LIN {X 0,Y 545.376,Z 587.4,A -85,B 0,C 180,E1 -3700.393,E2 -3700.393} C_VEL
LIN {X 0,Y 545.569,Z 576.596,A -85,B 0,C 180,E1 -3701.207,E2 -3701.207} C_VEL
LIN {X 0,Y 545.746,Z 565.176,A -85,B 0,C 180,E1 -3701.89,E2 -3701.89} C_VEL
LIN {X 0,Y 545.94,Z 552.979,A -85,B 0,C 180,E1 -3702.452,E2 -3702.452} C_VEL
LIN {X 0,Y 546.123,Z 540.184,A -85,B 0,C 180,E1 -3702.873,E2 -3702.873} C_VEL
LIN {X 0,Y 546.267,Z 526.619,A -85,B 0,C 180,E1 -3703.153,E2 -3703.153} C_VEL
LIN {X 0,Y 546.485,Z 429.804,A -85,B 0,C 180,E1 -3704.435,E2 -3704.435} C_VEL
LIN {X 0,Y 545.382,Z 422.607,A -85,B 0,C 180,E1 -3704.569,E2 -3704.569} C_VEL
LIN {X 0,Y 545.667,Z 401.74,A -85,B 0,C 180,E1 -3707.618,E2 -3707.618} C_VEL
LIN {X 0,Y 546.045,Z 380.777,A -85,B 0,C 180,E1 -3710.728,E2 -3710.728} C_VEL
LIN {X 0,Y 546.244,Z 365.01,A -85,B 0,C 180,E1 -3713.104,E2 -3713.104} C_VEL
LIN {X 0,Y 545.084,Z 358.59,A -85,B 0,C 180,E1 -3714.165,E2 -3714.165} C_VEL
LIN {X 0,Y 545.093,Z 358.583,A -85,B 0,C 180,E1 -3717.173,E2 -3717.173} C_VEL
LIN {X 0,Y 545.065,Z 358.589,A -85,B 0,C 180,E1 -3719.338,E2 -3719.338} C_VEL
LIN {X 0,Y 545.072,Z 358.591,A -85,B 0,C 180,E1 -3721.913,E2 -3721.913} C_VEL
LIN {X 0,Y 545.081,Z 358.582,A -85,B 0,C 180,E1 -3724.562,E2 -3724.562} C_VEL
LIN {X 0,Y 545.038,Z 358.591,A -85,B 0,C 180,E1 -3727.303,E2 -3727.303} C_VEL
LIN {X 0,Y 545.072,Z 358.585,A -85,B 0,C 180,E1 -3730.141,E2 -3730.141} C_VEL
LIN {X 0,Y 545.083,Z 358.584,A -85,B 0,C 180,E1 -3733.105,E2 -3733.105} C_VEL
LIN {X 0,Y 545.062,Z 358.585,A -85,B 0,C 180,E1 -3736.223,E2 -3736.223} C_VEL
LIN {X 0,Y 545.097,Z 358.581,A -85,B 0,C 180,E1 -3738.887,E2 -3738.887} C_VEL
LIN {X 0,Y 545.049,Z 358.591,A -85,B 0,C 180,E1 -3741.762,E2 -3741.762} C_VEL
LIN {X 0,Y 545.059,Z 358.585,A -85,B 0,C 180,E1 -3744.533,E2 -3744.533} C_VEL
LIN {X 0,Y 545.077,Z 358.589,A -85,B 0,C 180,E1 -3747.212,E2 -3747.212} C_VEL
LIN {X 0,Y 545.095,Z 358.583,A -85,B 0,C 180,E1 -3749.812,E2 -3749.812} C_VEL
LIN {X 0,Y 545.095,Z 358.583,A -85,B 0,C 180,E1 -3752.824,E2 -3752.824} C_VEL
LIN {X 0,Y 545.052,Z 358.59,A -85,B 0,C 180,E1 -3755.631,E2 -3755.631} C_VEL
LIN {X 0,Y 545.072,Z 358.583,A -85,B 0,C 180,E1 -3758.175,E2 -3758.175} C_VEL
LIN {X 0,Y 545.113,Z 358.578,A -85,B 0,C 180,E1 -3760.415,E2 -3760.415} C_VEL
LIN {X 0,Y 545.071,Z 358.587,A -85,B 0,C 180,E1 -3763.521,E2 -3763.521} C_VEL
LIN {X 0,Y 545.087,Z 358.582,A -85,B 0,C 180,E1 -3765.82,E2 -3765.82} C_VEL
LIN {X 0,Y 545.135,Z 358.581,A -85,B 0,C 180,E1 -3768.85,E2 -3768.85} C_VEL
LIN {X 0,Y 545.128,Z 358.576,A -85,B 0,C 180,E1 -3771.847,E2 -3771.847} C_VEL
LIN {X 0,Y 545.202,Z 358.573,A -85,B 0,C 180,E1 -3774.823,E2 -3774.823} C_VEL
LIN {X 0,Y 545.188,Z 358.569,A -85,B 0,C 180,E1 -3777.784,E2 -3777.784} C_VEL
LIN {X 0,Y 545.21,Z 358.572,A -85,B 0,C 180,E1 -3780.739,E2 -3780.739} C_VEL
LIN {X 0,Y 545.171,Z 358.579,A -85,B 0,C 180,E1 -3782.956,E2 -3782.956} C_VEL
LIN {X 0,Y 545.164,Z 358.571,A -85,B 0,C 180,E1 -3785.92,E2 -3785.92} C_VEL
LIN {X 0,Y 545.121,Z 358.585,A -85,B 0,C 180,E1 -3788.9,E2 -3788.9} C_VEL
LIN {X 0,Y 545.127,Z 358.576,A -85,B 0,C 180,E1 -3791.904,E2 -3791.904} C_VEL
LIN {X 0,Y 545.077,Z 358.589,A -85,B 0,C 180,E1 -3794.944,E2 -3794.944} C_VEL
LIN {X 0,Y 545.076,Z 358.584,A -85,B 0,C 180,E1 -3798.026,E2 -3798.026} C_VEL
LIN {X 0,Y 545.092,Z 358.586,A -85,B 0,C 180,E1 -3800.372,E2 -3800.372} C_VEL
LIN {X 0,Y 545.106,Z 358.579,A -85,B 0,C 180,E1 -3803.558,E2 -3803.558} C_VEL
LIN {X 0,Y 545.081,Z 358.583,A -85,B 0,C 180,E1 -3806.001,E2 -3806.001} C_VEL
LIN {X 0,Y 545.084,Z 358.588,A -85,B 0,C 180,E1 -3808.749,E2 -3808.749} C_VEL
LIN {X 0,Y 545.072,Z 358.583,A -85,B 0,C 180,E1 -3811.683,E2 -3811.683} C_VEL
LIN {X 0,Y 545.071,Z 358.591,A -85,B 0,C 180,E1 -3814.564,E2 -3814.564} C_VEL
LIN {X 0,Y 545.06,Z 358.586,A -85,B 0,C 180,E1 -3817.027,E2 -3817.027} C_VEL
LIN {X 0,Y 544.354,Z 358.673,A -85,B 0,C 180,E1 -3817.643,E2 -3817.643} C_VEL
LIN {X 0,Y 541.499,Z 359.034,A -85,B 0,C 180,E1 -3818.644,E2 -3818.644} C_VEL
LIN {X 0,Y 539.122,Z 359.327,A -85,B 0,C 180,E1 -3819.45,E2 -3819.45} C_VEL
LIN {X 0,Y 538.118,Z 359.454,A -85,B 0,C 180,E1 -3820.072,E2 -3820.072} C_VEL
LIN {X 0,Y 538.043,Z 359.459,A -85,B 0,C 180,E1 -3820.283,E2 -3820.283} C_VEL
LIN {X 0,Y 538.03,Z 359.461,A -85,B 0,C 180,E1 -3822.989,E2 -3822.989} C_VEL
LIN {X 0,Y 538.021,Z 359.465,A -85,B 0,C 180,E1 -3825.927,E2 -3825.927} C_VEL
LIN {X 0,Y 538.048,Z 359.458,A -85,B 0,C 180,E1 -3829.253,E2 -3829.253} C_VEL
LIN {X 0,Y 537.992,Z 359.473,A -85,B 0,C 180,E1 -3832.123,E2 -3832.123} C_VEL
LIN {X 0,Y 538.02,Z 359.462,A -85,B 0,C 180,E1 -3834.918,E2 -3834.918} C_VEL
LIN {X 0,Y 538.019,Z 359.464,A -85,B 0,C 180,E1 -3837.618,E2 -3837.618} C_VEL
LIN {X 0,Y 538.031,Z 359.468,A -85,B 0,C 180,E1 -3840.24,E2 -3840.24} C_VEL
LIN {X 0,Y 538.064,Z 359.457,A -85,B 0,C 180,E1 -3842.797,E2 -3842.797} C_VEL
LIN {X 0,Y 538.028,Z 359.463,A -85,B 0,C 180,E1 -3845.292,E2 -3845.292} C_VEL
LIN {X 0,Y 538.017,Z 359.472,A -85,B 0,C 180,E1 -3848.043,E2 -3848.043} C_VEL
LIN {X 0,Y 538.094,Z 359.486,A -85,B 0,C 180,E1 -3850.348,E2 -3850.348} C_VEL
LIN {X 0,Y 538.594,Z 365.48,A -85,B 0,C 180,E1 -3851.553,E2 -3851.553} C_VEL
LIN {X 0,Y 538.263,Z 380.54,A -85,B 0,C 180,E1 -3854.475,E2 -3854.475} C_VEL
LIN {X 0,Y 538.187,Z 384.837,A -85,B 0,C 180,E1 -3855.305,E2 -3855.305} C_VEL
LIN {X 0,Y 539.704,Z 393.756,A -85,B 0,C 180,E1 -3855.473,E2 -3855.473} C_VEL
LIN {X 0,Y 539.325,Z 491.401,A -85,B 0,C 180,E1 -3856.794,E2 -3856.794} C_VEL
LIN {X 0,Y 539.167,Z 504.592,A -85,B 0,C 180,E1 -3857.126,E2 -3857.126} C_VEL
LIN {X 0,Y 538.977,Z 516.69,A -85,B 0,C 180,E1 -3857.576,E2 -3857.576} C_VEL
LIN {X 0,Y 538.793,Z 528.843,A -85,B 0,C 180,E1 -3858.19,E2 -3858.19} C_VEL
LIN {X 0,Y 538.55,Z 539.767,A -85,B 0,C 180,E1 -3858.902,E2 -3858.902} C_VEL
LIN {X 0,Y 538.284,Z 550.235,A -85,B 0,C 180,E1 -3859.753,E2 -3859.753} C_VEL
LIN {X 0,Y 538.108,Z 558.785,A -85,B 0,C 180,E1 -3860.604,E2 -3860.604} C_VEL
LIN {X 0,Y 537.923,Z 566.658,A -85,B 0,C 180,E1 -3861.548,E2 -3861.548} C_VEL
LIN {X 0,Y 537.76,Z 574.357,A -85,B 0,C 180,E1 -3862.679,E2 -3862.679} C_VEL
LIN {X 0,Y 537.694,Z 581.463,A -85,B 0,C 180,E1 -3863.998,E2 -3863.998} C_VEL
LIN {X 0,Y 537.541,Z 586.202,A -85,B 0,C 180,E1 -3865.125,E2 -3865.125} C_VEL
LIN {X 0,Y 537.591,Z 589.833,A -85,B 0,C 180,E1 -3866.252,E2 -3866.252} C_VEL
LIN {X 0,Y 537.551,Z 591.71,A -85,B 0,C 180,E1 -3867.002,E2 -3867.002} C_VEL
LIN {X 0,Y 537.49,Z 593.128,A -85,B 0,C 180,E1 -3867.752,E2 -3867.752} C_VEL
LIN {X 0,Y 537.442,Z 594.757,A -85,B 0,C 180,E1 -3869.251,E2 -3869.251} C_VEL
LIN {X 0,Y 537.442,Z 594.996,A -85,B 0,C 180,E1 -3870,E2 -3870} C_VEL
LIN {X 0,Y 537.442,Z 594.814,A -85,B 0,C 180,E1 -3870.749,E2 -3870.749} C_VEL
LIN {X 0,Y 537.49,Z 593.26,A -85,B 0,C 180,E1 -3872.248,E2 -3872.248} C_VEL
LIN {X 0,Y 537.552,Z 591.899,A -85,B 0,C 180,E1 -3872.998,E2 -3872.998} C_VEL
LIN {X 0,Y 537.604,Z 589.022,A -85,B 0,C 180,E1 -3874.123,E2 -3874.123} C_VEL
LIN {X 0,Y 537.587,Z 585.12,A -85,B 0,C 180,E1 -3875.251,E2 -3875.251} C_VEL
LIN {X 0,Y 537.638,Z 580.368,A -85,B 0,C 180,E1 -3876.321,E2 -3876.321} C_VEL
LIN {X 0,Y 537.79,Z 573.76,A -85,B 0,C 180,E1 -3877.509,E2 -3877.509} C_VEL
LIN {X 0,Y 537.952,Z 565.884,A -85,B 0,C 180,E1 -3878.641,E2 -3878.641} C_VEL
LIN {X 0,Y 538.137,Z 556.083,A -85,B 0,C 180,E1 -3879.775,E2 -3879.775} C_VEL
LIN {X 0,Y 538.381,Z 545.805,A -85,B 0,C 180,E1 -3880.72,E2 -3880.72} C_VEL
LIN {X 0,Y 538.695,Z 534.835,A -85,B 0,C 180,E1 -3881.528,E2 -3881.528} C_VEL
LIN {X 0,Y 538.871,Z 524.477,A -85,B 0,C 180,E1 -3882.14,E2 -3882.14} C_VEL
LIN {X 0,Y 539.046,Z 511.974,A -85,B 0,C 180,E1 -3882.71,E2 -3882.71} C_VEL
LIN {X 0,Y 539.241,Z 498.545,A -85,B 0,C 180,E1 -3883.136,E2 -3883.136} C_VEL
LIN {X 0,Y 539.367,Z 485.208,A -85,B 0,C 180,E1 -3883.396,E2 -3883.396} C_VEL
LIN {X 0,Y 539.649,Z 393.1,A -85,B 0,C 180,E1 -3884.628,E2 -3884.628} C_VEL
LIN {X 0,Y 538.193,Z 384.795,A -85,B 0,C 180,E1 -3884.793,E2 -3884.793} C_VEL
LIN {X 0,Y 538.516,Z 368.756,A -85,B 0,C 180,E1 -3887.9,E2 -3887.9} C_VEL
LIN {X 0,Y 538.465,Z 361.938,A -85,B 0,C 180,E1 -3889.242,E2 -3889.242} C_VEL
LIN {X 0,Y 538.073,Z 359.464,A -85,B 0,C 180,E1 -3889.783,E2 -3889.783} C_VEL
LIN {X 0,Y 538.025,Z 359.465,A -85,B 0,C 180,E1 -3893.071,E2 -3893.071} C_VEL
LIN {X 0,Y 538.045,Z 359.465,A -85,B 0,C 180,E1 -3895.672,E2 -3895.672} C_VEL
LIN {X 0,Y 538.045,Z 359.467,A -85,B 0,C 180,E1 -3898.049,E2 -3898.049} C_VEL
LIN {X 0,Y 538.021,Z 359.462,A -85,B 0,C 180,E1 -3900.626,E2 -3900.626} C_VEL
LIN {X 0,Y 538.044,Z 359.46,A -85,B 0,C 180,E1 -3903.282,E2 -3903.282} C_VEL
LIN {X 0,Y 538.027,Z 359.468,A -85,B 0,C 180,E1 -3906.001,E2 -3906.001} C_VEL
LIN {X 0,Y 538.013,Z 359.462,A -85,B 0,C 180,E1 -3908.829,E2 -3908.829} C_VEL
LIN {X 0,Y 538.031,Z 359.47,A -85,B 0,C 180,E1 -3911.772,E2 -3911.772} C_VEL
LIN {X 0,Y 538.028,Z 359.461,A -85,B 0,C 180,E1 -3914.859,E2 -3914.859} C_VEL
LIN {X 0,Y 538.034,Z 359.463,A -85,B 0,C 180,E1 -3918.119,E2 -3918.119} C_VEL
LIN {X 0,Y 538.054,Z 359.458,A -85,B 0,C 180,E1 -3920.411,E2 -3920.411} C_VEL
LIN {X 0,Y 538.027,Z 359.462,A -85,B 0,C 180,E1 -3923.067,E2 -3923.067} C_VEL
LIN {X 0,Y 538.026,Z 359.466,A -85,B 0,C 180,E1 -3925.827,E2 -3925.827} C_VEL
LIN {X 0,Y 538.017,Z 359.462,A -85,B 0,C 180,E1 -3928.499,E2 -3928.499} C_VEL
LIN {X 0,Y 538.052,Z 359.461,A -85,B 0,C 180,E1 -3931.099,E2 -3931.099} C_VEL
LIN {X 0,Y 538.043,Z 359.466,A -85,B 0,C 180,E1 -3933.633,E2 -3933.633} C_VEL
LIN {X 0,Y 538.034,Z 359.461,A -85,B 0,C 180,E1 -3936.113,E2 -3936.113} C_VEL
LIN {X 0,Y 538.035,Z 359.469,A -85,B 0,C 180,E1 -3939.348,E2 -3939.348} C_VEL
LIN {X 0,Y 538.064,Z 359.456,A -85,B 0,C 180,E1 -3942.517,E2 -3942.517} C_VEL
LIN {X 0,Y 538.055,Z 359.462,A -85,B 0,C 180,E1 -3945.63,E2 -3945.63} C_VEL
LIN {X 0,Y 538.081,Z 359.456,A -85,B 0,C 180,E1 -3948.702,E2 -3948.702} C_VEL
LIN {X 0,Y 538.084,Z 359.456,A -85,B 0,C 180,E1 -3951.739,E2 -3951.739} C_VEL
LIN {X 0,Y 538.158,Z 359.447,A -85,B 0,C 180,E1 -3954.755,E2 -3954.755} C_VEL
LIN {X 0,Y 538.16,Z 359.445,A -85,B 0,C 180,E1 -3957.755,E2 -3957.755} C_VEL
LIN {X 0,Y 538.179,Z 359.446,A -85,B 0,C 180,E1 -3960.748,E2 -3960.748} C_VEL
LIN {X 0,Y 538.138,Z 359.455,A -85,B 0,C 180,E1 -3962.994,E2 -3962.994} C_VEL
LIN {X 0,Y 538.117,Z 359.449,A -85,B 0,C 180,E1 -3965.997,E2 -3965.997} C_VEL
LIN {X 0,Y 538.07,Z 359.464,A -85,B 0,C 180,E1 -3969.018,E2 -3969.018} C_VEL
LIN {X 0,Y 538.075,Z 359.455,A -85,B 0,C 180,E1 -3972.063,E2 -3972.063} C_VEL
LIN {X 0,Y 538.037,Z 359.465,A -85,B 0,C 180,E1 -3975.144,E2 -3975.144} C_VEL
LIN {X 0,Y 538.028,Z 359.462,A -85,B 0,C 180,E1 -3978.27,E2 -3978.27} C_VEL
LIN {X 0,Y 538.036,Z 359.466,A -85,B 0,C 180,E1 -3980.652,E2 -3980.652} C_VEL
LIN {X 0,Y 538.033,Z 359.46,A -85,B 0,C 180,E1 -3983.887,E2 -3983.887} C_VEL
LIN {X 0,Y 538.043,Z 359.463,A -85,B 0,C 180,E1 -3986.367,E2 -3986.367} C_VEL
LIN {X 0,Y 538.025,Z 359.466,A -85,B 0,C 180,E1 -3988.935,E2 -3988.935} C_VEL
LIN {X 0,Y 538.021,Z 359.462,A -85,B 0,C 180,E1 -3991.891,E2 -3991.891} C_VEL
LIN {X 0,Y 538.028,Z 359.47,A -85,B 0,C 180,E1 -3994.622,E2 -3994.622} C_VEL
LIN {X 0,Y 538.002,Z 359.465,A -85,B 0,C 180,E1 -3997.171,E2 -3997.171} C_VEL
LIN {X 0,Y 538.05,Z 359.458,A -85,B 0,C 180,E1 -3999.795,E2 -3999.795} C_VEL
LIN {X 0,Y 538.02,Z 359.466,A -85,B 0,C 180,E1 -4002.786,E2 -4002.786} C_VEL
LIN {X 0,Y 538.025,Z 359.463,A -85,B 0,C 180,E1 -4005.926,E2 -4005.926} C_VEL
LIN {X 0,Y 538.049,Z 359.458,A -85,B 0,C 180,E1 -4009.225,E2 -4009.225} C_VEL
LIN {X 0,Y 537.992,Z 359.471,A -85,B 0,C 180,E1 -4012.123,E2 -4012.123} C_VEL
LIN {X 0,Y 538.02,Z 359.463,A -85,B 0,C 180,E1 -4014.918,E2 -4014.918} C_VEL
LIN {X 0,Y 538.031,Z 359.461,A -85,B 0,C 180,E1 -4017.619,E2 -4017.619} C_VEL
LIN {X 0,Y 538.018,Z 359.471,A -85,B 0,C 180,E1 -4020.24,E2 -4020.24} C_VEL
LIN {X 0,Y 538.063,Z 359.461,A -85,B 0,C 180,E1 -4022.797,E2 -4022.797} C_VEL
LIN {X 0,Y 538.066,Z 359.506,A -85,B 0,C 180,E1 -4025.706,E2 -4025.706} C_VEL
LIN {X 0,Y 539.402,Z 367.417,A -85,B 0,C 180,E1 -4026.991,E2 -4026.991} C_VEL
LIN {X 0,Y 538.969,Z 387.025,A -85,B 0,C 180,E1 -4029.973,E2 -4029.973} C_VEL
LIN {X 0,Y 538.622,Z 405.421,A -85,B 0,C 180,E1 -4032.732,E2 -4032.732} C_VEL
LIN {X 0,Y 538.361,Z 422.372,A -85,B 0,C 180,E1 -4035.239,E2 -4035.239} C_VEL
LIN {X 0,Y 539.666,Z 431.29,A -85,B 0,C 180,E1 -4035.403,E2 -4035.403} C_VEL
LIN {X 0,Y 539.307,Z 530.771,A -85,B 0,C 180,E1 -4036.746,E2 -4036.746} C_VEL
LIN {X 0,Y 539.172,Z 544.06,A -85,B 0,C 180,E1 -4037.078,E2 -4037.078} C_VEL
LIN {X 0,Y 538.946,Z 556.237,A -85,B 0,C 180,E1 -4037.527,E2 -4037.527} C_VEL
LIN {X 0,Y 538.691,Z 568.091,A -85,B 0,C 180,E1 -4038.117,E2 -4038.117} C_VEL
LIN {X 0,Y 538.499,Z 580.143,A -85,B 0,C 180,E1 -4038.901,E2 -4038.901} C_VEL
LIN {X 0,Y 538.263,Z 590.602,A -85,B 0,C 180,E1 -4039.753,E2 -4039.753} C_VEL
LIN {X 0,Y 538.067,Z 599.115,A -85,B 0,C 180,E1 -4040.603,E2 -4040.603} C_VEL
LIN {X 0,Y 537.921,Z 606.962,A -85,B 0,C 180,E1 -4041.548,E2 -4041.548} C_VEL
LIN {X 0,Y 537.754,Z 614.622,A -85,B 0,C 180,E1 -4042.679,E2 -4042.679} C_VEL
LIN {X 0,Y 537.693,Z 621.68,A -85,B 0,C 180,E1 -4043.998,E2 -4043.998} C_VEL
LIN {X 0,Y 537.54,Z 626.373,A -85,B 0,C 180,E1 -4045.125,E2 -4045.125} C_VEL
LIN {X 0,Y 537.591,Z 629.958,A -85,B 0,C 180,E1 -4046.252,E2 -4046.252} C_VEL
LIN {X 0,Y 537.551,Z 631.807,A -85,B 0,C 180,E1 -4047.002,E2 -4047.002} C_VEL
LIN {X 0,Y 537.451,Z 634.182,A -85,B 0,C 180,E1 -4048.501,E2 -4048.501} C_VEL
LIN {X 0,Y 537.442,Z 635,A -85,B 0,C 180,E1 -4050,E2 -4050} C_VEL
LIN {X 0,Y 537.451,Z 634.184,A -85,B 0,C 180,E1 -4051.499,E2 -4051.499} C_VEL
LIN {X 0,Y 537.551,Z 631.81,A -85,B 0,C 180,E1 -4052.998,E2 -4052.998} C_VEL
LIN {X 0,Y 537.603,Z 628.895,A -85,B 0,C 180,E1 -4054.123,E2 -4054.123} C_VEL
LIN {X 0,Y 537.588,Z 624.948,A -85,B 0,C 180,E1 -4055.251,E2 -4055.251} C_VEL
LIN {X 0,Y 537.644,Z 620.125,A -85,B 0,C 180,E1 -4056.326,E2 -4056.326} C_VEL
LIN {X 0,Y 537.79,Z 613.467,A -85,B 0,C 180,E1 -4057.509,E2 -4057.509} C_VEL
LIN {X 0,Y 537.972,Z 605.478,A -85,B 0,C 180,E1 -4058.64,E2 -4058.64} C_VEL
LIN {X 0,Y 538.143,Z 597.335,A -85,B 0,C 180,E1 -4059.585,E2 -4059.585} C_VEL
LIN {X 0,Y 538.383,Z 587.382,A -85,B 0,C 180,E1 -4060.53,E2 -4060.53} C_VEL
LIN {X 0,Y 538.565,Z 577.533,A -85,B 0,C 180,E1 -4061.288,E2 -4061.288} C_VEL
LIN {X 0,Y 538.731,Z 566.441,A -85,B 0,C 180,E1 -4061.973,E2 -4061.973} C_VEL
LIN {X 0,Y 538.948,Z 553.962,A -85,B 0,C 180,E1 -4062.568,E2 -4062.568} C_VEL
LIN {X 0,Y 539.189,Z 540.923,A -85,B 0,C 180,E1 -4063.017,E2 -4063.017} C_VEL
LIN {X 0,Y 539.369,Z 527.931,A -85,B 0,C 180,E1 -4063.3,E2 -4063.3} C_VEL
LIN {X 0,Y 539.581,Z 430.466,A -85,B 0,C 180,E1 -4064.611,E2 -4064.611} C_VEL
LIN {X 0,Y 538.377,Z 422.337,A -85,B 0,C 180,E1 -4064.767,E2 -4064.767} C_VEL
LIN {X 0,Y 538.748,Z 399.913,A -85,B 0,C 180,E1 -4068.088,E2 -4068.088} C_VEL
LIN {X 0,Y 539.145,Z 379.235,A -85,B 0,C 180,E1 -4071.206,E2 -4071.206} C_VEL
LIN {X 0,Y 539.284,Z 366.092,A -85,B 0,C 180,E1 -4073.217,E2 -4073.217} C_VEL
LIN {X 0,Y 538.034,Z 359.468,A -85,B 0,C 180,E1 -4074.322,E2 -4074.322} C_VEL
LIN {X 0,Y 538.063,Z 359.459,A -85,B 0,C 180,E1 -4077.203,E2 -4077.203} C_VEL
LIN {X 0,Y 538.018,Z 359.471,A -85,B 0,C 180,E1 -4079.76,E2 -4079.76} C_VEL
LIN {X 0,Y 538.031,Z 359.461,A -85,B 0,C 180,E1 -4082.381,E2 -4082.381} C_VEL
LIN {X 0,Y 538.02,Z 359.463,A -85,B 0,C 180,E1 -4085.082,E2 -4085.082} C_VEL
LIN {X 0,Y 537.992,Z 359.471,A -85,B 0,C 180,E1 -4087.877,E2 -4087.877} C_VEL
LIN {X 0,Y 538.049,Z 359.458,A -85,B 0,C 180,E1 -4090.775,E2 -4090.775} C_VEL
LIN {X 0,Y 538.025,Z 359.463,A -85,B 0,C 180,E1 -4094.074,E2 -4094.074} C_VEL
LIN {X 0,Y 538.02,Z 359.466,A -85,B 0,C 180,E1 -4097.214,E2 -4097.214} C_VEL
LIN {X 0,Y 538.05,Z 359.458,A -85,B 0,C 180,E1 -4100.205,E2 -4100.205} C_VEL
LIN {X 0,Y 538.023,Z 359.465,A -85,B 0,C 180,E1 -4103.067,E2 -4103.067} C_VEL
LIN {X 0,Y 538.026,Z 359.464,A -85,B 0,C 180,E1 -4105.827,E2 -4105.827} C_VEL
LIN {X 0,Y 538.017,Z 359.462,A -85,B 0,C 180,E1 -4108.499,E2 -4108.499} C_VEL
LIN {X 0,Y 538.052,Z 359.463,A -85,B 0,C 180,E1 -4111.099,E2 -4111.099} C_VEL
LIN {X 0,Y 538.043,Z 359.463,A -85,B 0,C 180,E1 -4113.633,E2 -4113.633} C_VEL
LIN {X 0,Y 538.033,Z 359.46,A -85,B 0,C 180,E1 -4116.113,E2 -4116.113} C_VEL
LIN {X 0,Y 538.036,Z 359.467,A -85,B 0,C 180,E1 -4119.348,E2 -4119.348} C_VEL
LIN {X 0,Y 538.064,Z 359.457,A -85,B 0,C 180,E1 -4122.517,E2 -4122.517} C_VEL
LIN {X 0,Y 538.055,Z 359.46,A -85,B 0,C 180,E1 -4125.63,E2 -4125.63} C_VEL
LIN {X 0,Y 538.089,Z 359.457,A -85,B 0,C 180,E1 -4128.702,E2 -4128.702} C_VEL
LIN {X 0,Y 538.084,Z 359.454,A -85,B 0,C 180,E1 -4131.74,E2 -4131.74} C_VEL
LIN {X 0,Y 538.158,Z 359.45,A -85,B 0,C 180,E1 -4134.755,E2 -4134.755} C_VEL
LIN {X 0,Y 538.16,Z 359.444,A -85,B 0,C 180,E1 -4137.755,E2 -4137.755} C_VEL
LIN {X 0,Y 538.18,Z 359.448,A -85,B 0,C 180,E1 -4140.748,E2 -4140.748} C_VEL
LIN {X 0,Y 538.137,Z 359.455,A -85,B 0,C 180,E1 -4142.995,E2 -4142.995} C_VEL
LIN {X 0,Y 538.117,Z 359.45,A -85,B 0,C 180,E1 -4145.997,E2 -4145.997} C_VEL
LIN {X 0,Y 538.07,Z 359.462,A -85,B 0,C 180,E1 -4149.018,E2 -4149.018} C_VEL
LIN {X 0,Y 538.075,Z 359.455,A -85,B 0,C 180,E1 -4152.063,E2 -4152.063} C_VEL
LIN {X 0,Y 538.037,Z 359.463,A -85,B 0,C 180,E1 -4155.144,E2 -4155.144} C_VEL
LIN {X 0,Y 538.028,Z 359.464,A -85,B 0,C 180,E1 -4158.27,E2 -4158.27} C_VEL
LIN {X 0,Y 538.035,Z 359.469,A -85,B 0,C 180,E1 -4160.652,E2 -4160.652} C_VEL
LIN {X 0,Y 538.034,Z 359.46,A -85,B 0,C 180,E1 -4163.887,E2 -4163.887} C_VEL
LIN {X 0,Y 538.043,Z 359.465,A -85,B 0,C 180,E1 -4166.367,E2 -4166.367} C_VEL
LIN {X 0,Y 538.025,Z 359.464,A -85,B 0,C 180,E1 -4168.935,E2 -4168.935} C_VEL
LIN {X 0,Y 538.021,Z 359.463,A -85,B 0,C 180,E1 -4171.891,E2 -4171.891} C_VEL
LIN {X 0,Y 538.02,Z 359.469,A -85,B 0,C 180,E1 -4174.621,E2 -4174.621} C_VEL
LIN {X 0,Y 538.004,Z 359.464,A -85,B 0,C 180,E1 -4177.171,E2 -4177.171} C_VEL
LIN {X 0,Y 538.043,Z 359.459,A -85,B 0,C 180,E1 -4180.283,E2 -4180.283} C_VEL
LIN {X 0,Y 537.392,Z 359.543,A -85,B 0,C 180,E1 -4180.908,E2 -4180.908} C_VEL
LIN {X 0,Y 534.533,Z 359.899,A -85,B 0,C 180,E1 -4181.922,E2 -4181.922} C_VEL
LIN {X 0,Y 532.1,Z 360.203,A -85,B 0,C 180,E1 -4182.739,E2 -4182.739} C_VEL
LIN {X 0,Y 531.048,Z 360.33,A -85,B 0,C 180,E1 -4183.37,E2 -4183.37} C_VEL
LIN {X 0,Y 530.96,Z 360.341,A -85,B 0,C 180,E1 -4183.584,E2 -4183.584} C_VEL
LIN {X 0,Y 530.955,Z 360.348,A -85,B 0,C 180,E1 -4186.506,E2 -4186.506} C_VEL
LIN {X 0,Y 530.984,Z 360.339,A -85,B 0,C 180,E1 -4188.977,E2 -4188.977} C_VEL
LIN {X 0,Y 530.957,Z 360.342,A -85,B 0,C 180,E1 -4191.53,E2 -4191.53} C_VEL
LIN {X 0,Y 530.981,Z 360.345,A -85,B 0,C 180,E1 -4194.383,E2 -4194.383} C_VEL
LIN {X 0,Y 530.966,Z 360.34,A -85,B 0,C 180,E1 -4197.134,E2 -4197.134} C_VEL
LIN {X 0,Y 530.982,Z 360.343,A -85,B 0,C 180,E1 -4199.805,E2 -4199.805} C_VEL
LIN {X 0,Y 531.016,Z 360.338,A -85,B 0,C 180,E1 -4202.468,E2 -4202.468} C_VEL
LIN {X 0,Y 530.996,Z 360.339,A -85,B 0,C 180,E1 -4204.943,E2 -4204.943} C_VEL
LIN {X 0,Y 530.973,Z 360.348,A -85,B 0,C 180,E1 -4208.247,E2 -4208.247} C_VEL
LIN {X 0,Y 531.079,Z 360.457,A -85,B 0,C 180,E1 -4210.23,E2 -4210.23} C_VEL
LIN {X 0,Y 531.615,Z 366.698,A -85,B 0,C 180,E1 -4211.502,E2 -4211.502} C_VEL
LIN {X 0,Y 531.245,Z 382.781,A -85,B 0,C 180,E1 -4214.658,E2 -4214.658} C_VEL
LIN {X 0,Y 531.21,Z 385.047,A -85,B 0,C 180,E1 -4215.099,E2 -4215.099} C_VEL
LIN {X 0,Y 532.835,Z 394.046,A -85,B 0,C 180,E1 -4215.281,E2 -4215.281} C_VEL
LIN {X 0,Y 532.421,Z 491.697,A -85,B 0,C 180,E1 -4216.62,E2 -4216.62} C_VEL
LIN {X 0,Y 532.271,Z 504.877,A -85,B 0,C 180,E1 -4216.956,E2 -4216.956} C_VEL
LIN {X 0,Y 532.061,Z 516.971,A -85,B 0,C 180,E1 -4217.412,E2 -4217.412} C_VEL
LIN {X 0,Y 531.873,Z 528.75,A -85,B 0,C 180,E1 -4218.011,E2 -4218.011} C_VEL
LIN {X 0,Y 531.591,Z 540.042,A -85,B 0,C 180,E1 -4218.755,E2 -4218.755} C_VEL
LIN {X 0,Y 531.298,Z 550.509,A -85,B 0,C 180,E1 -4219.617,E2 -4219.617} C_VEL
LIN {X 0,Y 531.102,Z 559.058,A -85,B 0,C 180,E1 -4220.479,E2 -4220.479} C_VEL
LIN {X 0,Y 530.906,Z 566.93,A -85,B 0,C 180,E1 -4221.436,E2 -4221.436} C_VEL
LIN {X 0,Y 530.723,Z 574.627,A -85,B 0,C 180,E1 -4222.582,E2 -4222.582} C_VEL
LIN {X 0,Y 530.63,Z 581.682,A -85,B 0,C 180,E1 -4223.918,E2 -4223.918} C_VEL
LIN {X 0,Y 530.459,Z 586.389,A -85,B 0,C 180,E1 -4225.06,E2 -4225.06} C_VEL
LIN {X 0,Y 530.516,Z 589.987,A -85,B 0,C 180,E1 -4226.202,E2 -4226.202} C_VEL
LIN {X 0,Y 530.457,Z 591.851,A -85,B 0,C 180,E1 -4226.962,E2 -4226.962} C_VEL
LIN {X 0,Y 530.411,Z 593.257,A -85,B 0,C 180,E1 -4227.722,E2 -4227.722} C_VEL
LIN {X 0,Y 530.344,Z 594.874,A -85,B 0,C 180,E1 -4229.241,E2 -4229.241} C_VEL
LIN {X 0,Y 530.344,Z 595.112,A -85,B 0,C 180,E1 -4230,E2 -4230} C_VEL
LIN {X 0,Y 530.344,Z 594.93,A -85,B 0,C 180,E1 -4230.759,E2 -4230.759} C_VEL
LIN {X 0,Y 530.411,Z 593.386,A -85,B 0,C 180,E1 -4232.278,E2 -4232.278} C_VEL
LIN {X 0,Y 530.457,Z 592.035,A -85,B 0,C 180,E1 -4233.038,E2 -4233.038} C_VEL
LIN {X 0,Y 530.523,Z 589.18,A -85,B 0,C 180,E1 -4234.178,E2 -4234.178} C_VEL
LIN {X 0,Y 530.524,Z 585.31,A -85,B 0,C 180,E1 -4235.321,E2 -4235.321} C_VEL
LIN {X 0,Y 530.622,Z 579.62,A -85,B 0,C 180,E1 -4236.603,E2 -4236.603} C_VEL
LIN {X 0,Y 530.779,Z 572.803,A -85,B 0,C 180,E1 -4237.8,E2 -4237.8} C_VEL
LIN {X 0,Y 530.922,Z 564.672,A -85,B 0,C 180,E1 -4238.948,E2 -4238.948} C_VEL
LIN {X 0,Y 531.131,Z 556.345,A -85,B 0,C 180,E1 -4239.905,E2 -4239.905} C_VEL
LIN {X 0,Y 531.407,Z 546.065,A -85,B 0,C 180,E1 -4240.863,E2 -4240.863} C_VEL
LIN {X 0,Y 531.732,Z 535.506,A -85,B 0,C 180,E1 -4241.653,E2 -4241.653} C_VEL
LIN {X 0,Y 531.935,Z 524.732,A -85,B 0,C 180,E1 -4242.301,E2 -4242.301} C_VEL
LIN {X 0,Y 532.127,Z 513.439,A -85,B 0,C 180,E1 -4242.829,E2 -4242.829} C_VEL
LIN {X 0,Y 532.323,Z 500.616,A -85,B 0,C 180,E1 -4243.261,E2 -4243.261} C_VEL
LIN {X 0,Y 532.499,Z 486.969,A -85,B 0,C 180,E1 -4243.548,E2 -4243.548} C_VEL
LIN {X 0,Y 532.79,Z 394.069,A -85,B 0,C 180,E1 -4244.81,E2 -4244.81} C_VEL
LIN {X 0,Y 531.204,Z 385.087,A -85,B 0,C 180,E1 -4244.981,E2 -4244.981} C_VEL
LIN {X 0,Y 531.542,Z 369.374,A -85,B 0,C 180,E1 -4248.062,E2 -4248.062} C_VEL
LIN {X 0,Y 531.498,Z 363.144,A -85,B 0,C 180,E1 -4249.303,E2 -4249.303} C_VEL
LIN {X 0,Y 531.037,Z 360.341,A -85,B 0,C 180,E1 -4249.912,E2 -4249.912} C_VEL
LIN {X 0,Y 530.952,Z 360.349,A -85,B 0,C 180,E1 -4252.573,E2 -4252.573} C_VEL
LIN {X 0,Y 531.007,Z 360.338,A -85,B 0,C 180,E1 -4255.057,E2 -4255.057} C_VEL
LIN {X 0,Y 531.016,Z 360.337,A -85,B 0,C 180,E1 -4257.595,E2 -4257.595} C_VEL
LIN {X 0,Y 530.974,Z 360.34,A -85,B 0,C 180,E1 -4260.644,E2 -4260.644} C_VEL
LIN {X 0,Y 530.99,Z 360.344,A -85,B 0,C 180,E1 -4263.772,E2 -4263.772} C_VEL
LIN {X 0,Y 530.967,Z 360.341,A -85,B 0,C 180,E1 -4266.557,E2 -4266.557} C_VEL
LIN {X 0,Y 530.982,Z 360.347,A -85,B 0,C 180,E1 -4269.854,E2 -4269.854} C_VEL
LIN {X 0,Y 530.975,Z 360.34,A -85,B 0,C 180,E1 -4272.456,E2 -4272.456} C_VEL
LIN {X 0,Y 530.984,Z 360.346,A -85,B 0,C 180,E1 -4275.62,E2 -4275.62} C_VEL
LIN {X 0,Y 531.003,Z 360.336,A -85,B 0,C 180,E1 -4278.565,E2 -4278.565} C_VEL
LIN {X 0,Y 530.964,Z 360.345,A -85,B 0,C 180,E1 -4281.345,E2 -4281.345} C_VEL
LIN {X 0,Y 530.977,Z 360.339,A -85,B 0,C 180,E1 -4284.381,E2 -4284.381} C_VEL
LIN {X 0,Y 530.969,Z 360.343,A -85,B 0,C 180,E1 -4287.133,E2 -4287.133} C_VEL
LIN {X 0,Y 530.963,Z 360.346,A -85,B 0,C 180,E1 -4289.802,E2 -4289.802} C_VEL
LIN {X 0,Y 531.01,Z 360.335,A -85,B 0,C 180,E1 -4292.466,E2 -4292.466} C_VEL
LIN {X 0,Y 531.002,Z 360.338,A -85,B 0,C 180,E1 -4294.942,E2 -4294.942} C_VEL
LIN {X 0,Y 530.984,Z 360.341,A -85,B 0,C 180,E1 -4297.893,E2 -4297.893} C_VEL
LIN {X 0,Y 530.989,Z 360.338,A -85,B 0,C 180,E1 -4300.677,E2 -4300.677} C_VEL
LIN {X 0,Y 530.986,Z 360.343,A -85,B 0,C 180,E1 -4303.071,E2 -4303.071} C_VEL
LIN {X 0,Y 531.031,Z 360.34,A -85,B 0,C 180,E1 -4305.436,E2 -4305.436} C_VEL
LIN {X 0,Y 531.038,Z 360.332,A -85,B 0,C 180,E1 -4308.55,E2 -4308.55} C_VEL
LIN {X 0,Y 531.052,Z 360.333,A -85,B 0,C 180,E1 -4311.629,E2 -4311.629} C_VEL
LIN {X 0,Y 531.117,Z 360.324,A -85,B 0,C 180,E1 -4314.685,E2 -4314.685} C_VEL
LIN {X 0,Y 531.132,Z 360.321,A -85,B 0,C 180,E1 -4317.725,E2 -4317.725} C_VEL
LIN {X 0,Y 531.148,Z 360.322,A -85,B 0,C 180,E1 -4320.758,E2 -4320.758} C_VEL
LIN {X 0,Y 531.104,Z 360.332,A -85,B 0,C 180,E1 -4323.034,E2 -4323.034} C_VEL
LIN {X 0,Y 531.076,Z 360.326,A -85,B 0,C 180,E1 -4326.077,E2 -4326.077} C_VEL
LIN {X 0,Y 531.03,Z 360.339,A -85,B 0,C 180,E1 -4329.138,E2 -4329.138} C_VEL
LIN {X 0,Y 531.052,Z 360.33,A -85,B 0,C 180,E1 -4331.678,E2 -4331.678} C_VEL
LIN {X 0,Y 531.021,Z 360.342,A -85,B 0,C 180,E1 -4334.956,E2 -4334.956} C_VEL
LIN {X 0,Y 531.008,Z 360.335,A -85,B 0,C 180,E1 -4337.723,E2 -4337.723} C_VEL
LIN {X 0,Y 530.998,Z 360.344,A -85,B 0,C 180,E1 -4340.938,E2 -4340.938} C_VEL
LIN {X 0,Y 531,Z 360.337,A -85,B 0,C 180,E1 -4344.046,E2 -4344.046} C_VEL
LIN {X 0,Y 531.005,Z 360.345,A -85,B 0,C 180,E1 -4346.744,E2 -4346.744} C_VEL
LIN {X 0,Y 530.976,Z 360.34,A -85,B 0,C 180,E1 -4349.323,E2 -4349.323} C_VEL
LIN {X 0,Y 530.974,Z 360.341,A -85,B 0,C 180,E1 -4352.104,E2 -4352.104} C_VEL
LIN {X 0,Y 530.985,Z 360.343,A -85,B 0,C 180,E1 -4354.855,E2 -4354.855} C_VEL
LIN {X 0,Y 530.961,Z 360.341,A -85,B 0,C 180,E1 -4357.508,E2 -4357.508} C_VEL
LIN {X 0,Y 531.021,Z 360.341,A -85,B 0,C 180,E1 -4360.429,E2 -4360.429} C_VEL
LIN {X 0,Y 530.963,Z 360.341,A -85,B 0,C 180,E1 -4363.495,E2 -4363.495} C_VEL
LIN {X 0,Y 530.963,Z 360.349,A -85,B 0,C 180,E1 -4366.506,E2 -4366.506} C_VEL
LIN {X 0,Y 530.986,Z 360.339,A -85,B 0,C 180,E1 -4368.976,E2 -4368.976} C_VEL
LIN {X 0,Y 530.957,Z 360.342,A -85,B 0,C 180,E1 -4371.53,E2 -4371.53} C_VEL
LIN {X 0,Y 530.981,Z 360.347,A -85,B 0,C 180,E1 -4374.383,E2 -4374.383} C_VEL
LIN {X 0,Y 530.972,Z 360.34,A -85,B 0,C 180,E1 -4377.135,E2 -4377.135} C_VEL
LIN {X 0,Y 530.97,Z 360.343,A -85,B 0,C 180,E1 -4379.804,E2 -4379.804} C_VEL
LIN {X 0,Y 531.015,Z 360.342,A -85,B 0,C 180,E1 -4382.468,E2 -4382.468} C_VEL
LIN {X 0,Y 531.014,Z 360.418,A -85,B 0,C 180,E1 -4385.544,E2 -4385.544} C_VEL
LIN {X 0,Y 532.447,Z 368.495,A -85,B 0,C 180,E1 -4386.879,E2 -4386.879} C_VEL
LIN {X 0,Y 532.008,Z 388.171,A -85,B 0,C 180,E1 -4389.912,E2 -4389.912} C_VEL
LIN {X 0,Y 531.57,Z 407.794,A -85,B 0,C 180,E1 -4392.893,E2 -4392.893} C_VEL
LIN {X 0,Y 531.347,Z 422.302,A -85,B 0,C 180,E1 -4395.05,E2 -4395.05} C_VEL
LIN {X 0,Y 532.8,Z 433.007,A -85,B 0,C 180,E1 -4395.237,E2 -4395.237} C_VEL
LIN {X 0,Y 532.404,Z 530.504,A -85,B 0,C 180,E1 -4396.571,E2 -4396.571} C_VEL
LIN {X 0,Y 532.24,Z 543.792,A -85,B 0,C 180,E1 -4396.907,E2 -4396.907} C_VEL
LIN {X 0,Y 531.987,Z 555.968,A -85,B 0,C 180,E1 -4397.361,E2 -4397.361} C_VEL
LIN {X 0,Y 531.724,Z 568.243,A -85,B 0,C 180,E1 -4397.984,E2 -4397.984} C_VEL
LIN {X 0,Y 531.512,Z 579.875,A -85,B 0,C 180,E1 -4398.754,E2 -4398.754} C_VEL
LIN {X 0,Y 531.22,Z 590.334,A -85,B 0,C 180,E1 -4399.615,E2 -4399.615} C_VEL
LIN {X 0,Y 531.033,Z 598.888,A -85,B 0,C 180,E1 -4400.478,E2 -4400.478} C_VEL
LIN {X 0,Y 530.886,Z 606.784,A -85,B 0,C 180,E1 -4401.435,E2 -4401.435} C_VEL
LIN {X 0,Y 530.681,Z 614.493,A -85,B 0,C 180,E1 -4402.581,E2 -4402.581} C_VEL
LIN {X 0,Y 530.604,Z 621.603,A -85,B 0,C 180,E1 -4403.918,E2 -4403.918} C_VEL
LIN {X 0,Y 530.459,Z 626.33,A -85,B 0,C 180,E1 -4405.06,E2 -4405.06} C_VEL
LIN {X 0,Y 530.516,Z 629.947,A -85,B 0,C 180,E1 -4406.202,E2 -4406.202} C_VEL
LIN {X 0,Y 530.457,Z 631.804,A -85,B 0,C 180,E1 -4406.962,E2 -4406.962} C_VEL
LIN {X 0,Y 530.41,Z 633.192,A -85,B 0,C 180,E1 -4407.722,E2 -4407.722} C_VEL
LIN {X 0,Y 530.344,Z 634.785,A -85,B 0,C 180,E1 -4409.241,E2 -4409.241} C_VEL
LIN {X 0,Y 530.342,Z 635,A -85,B 0,C 180,E1 -4410,E2 -4410} C_VEL
LIN {X 0,Y 530.361,Z 634.183,A -85,B 0,C 180,E1 -4411.519,E2 -4411.519} C_VEL
LIN {X 0,Y 530.41,Z 633.195,A -85,B 0,C 180,E1 -4412.278,E2 -4412.278} C_VEL
LIN {X 0,Y 530.457,Z 631.807,A -85,B 0,C 180,E1 -4413.038,E2 -4413.038} C_VEL
LIN {X 0,Y 530.522,Z 628.876,A -85,B 0,C 180,E1 -4414.178,E2 -4414.178} C_VEL
LIN {X 0,Y 530.525,Z 624.896,A -85,B 0,C 180,E1 -4415.321,E2 -4415.321} C_VEL
LIN {X 0,Y 530.596,Z 619.183,A -85,B 0,C 180,E1 -4416.579,E2 -4416.579} C_VEL
LIN {X 0,Y 530.735,Z 612.091,A -85,B 0,C 180,E1 -4417.801,E2 -4417.801} C_VEL
LIN {X 0,Y 530.93,Z 603.796,A -85,B 0,C 180,E1 -4418.948,E2 -4418.948} C_VEL
LIN {X 0,Y 531.126,Z 595.296,A -85,B 0,C 180,E1 -4419.905,E2 -4419.905} C_VEL
LIN {X 0,Y 531.38,Z 584.795,A -85,B 0,C 180,E1 -4420.863,E2 -4420.863} C_VEL
LIN {X 0,Y 531.662,Z 572.834,A -85,B 0,C 180,E1 -4421.736,E2 -4421.736} C_VEL
LIN {X 0,Y 531.948,Z 561.102,A -85,B 0,C 180,E1 -4422.397,E2 -4422.397} C_VEL
LIN {X 0,Y 532.166,Z 548.748,A -85,B 0,C 180,E1 -4422.925,E2 -4422.925} C_VEL
LIN {X 0,Y 532.342,Z 536.078,A -85,B 0,C 180,E1 -4423.309,E2 -4423.309} C_VEL
LIN {X 0,Y 532.492,Z 522.869,A -85,B 0,C 180,E1 -4423.548,E2 -4423.548} C_VEL
LIN {X 0,Y 532.706,Z 431.188,A -85,B 0,C 180,E1 -4424.79,E2 -4424.79} C_VEL
LIN {X 0,Y 531.333,Z 422.114,A -85,B 0,C 180,E1 -4424.963,E2 -4424.963} C_VEL
LIN {X 0,Y 531.737,Z 401.066,A -85,B 0,C 180,E1 -4428.122,E2 -4428.122} C_VEL
LIN {X 0,Y 532.193,Z 380.313,A -85,B 0,C 180,E1 -4431.294,E2 -4431.294} C_VEL
LIN {X 0,Y 532.446,Z 368.493,A -85,B 0,C 180,E1 -4433.121,E2 -4433.121} C_VEL
LIN {X 0,Y 530.997,Z 360.343,A -85,B 0,C 180,E1 -4434.483,E2 -4434.483} C_VEL
LIN {X 0,Y 531.015,Z 360.342,A -85,B 0,C 180,E1 -4437.532,E2 -4437.532} C_VEL
LIN {X 0,Y 530.974,Z 360.341,A -85,B 0,C 180,E1 -4440.645,E2 -4440.645} C_VEL
LIN {X 0,Y 530.99,Z 360.346,A -85,B 0,C 180,E1 -4443.772,E2 -4443.772} C_VEL
LIN {X 0,Y 530.967,Z 360.34,A -85,B 0,C 180,E1 -4446.557,E2 -4446.557} C_VEL
LIN {X 0,Y 530.982,Z 360.344,A -85,B 0,C 180,E1 -4449.854,E2 -4449.854} C_VEL
LIN {X 0,Y 530.979,Z 360.339,A -85,B 0,C 180,E1 -4452.455,E2 -4452.455} C_VEL
LIN {X 0,Y 530.984,Z 360.346,A -85,B 0,C 180,E1 -4455.62,E2 -4455.62} C_VEL
LIN {X 0,Y 531.003,Z 360.336,A -85,B 0,C 180,E1 -4458.565,E2 -4458.565} C_VEL
LIN {X 0,Y 530.964,Z 360.348,A -85,B 0,C 180,E1 -4461.345,E2 -4461.345} C_VEL
LIN {X 0,Y 530.976,Z 360.339,A -85,B 0,C 180,E1 -4464.382,E2 -4464.382} C_VEL
LIN {X 0,Y 530.969,Z 360.345,A -85,B 0,C 180,E1 -4467.133,E2 -4467.133} C_VEL
LIN {X 0,Y 530.979,Z 360.341,A -85,B 0,C 180,E1 -4469.804,E2 -4469.804} C_VEL
LIN {X 0,Y 531.01,Z 360.335,A -85,B 0,C 180,E1 -4472.466,E2 -4472.466} C_VEL
LIN {X 0,Y 531.002,Z 360.34,A -85,B 0,C 180,E1 -4474.942,E2 -4474.942} C_VEL
LIN {X 0,Y 530.984,Z 360.339,A -85,B 0,C 180,E1 -4477.893,E2 -4477.893} C_VEL
LIN {X 0,Y 530.989,Z 360.339,A -85,B 0,C 180,E1 -4480.677,E2 -4480.677} C_VEL
LIN {X 0,Y 530.986,Z 360.346,A -85,B 0,C 180,E1 -4483.071,E2 -4483.071} C_VEL
LIN {X 0,Y 531.01,Z 360.34,A -85,B 0,C 180,E1 -4485.436,E2 -4485.436} C_VEL
LIN {X 0,Y 531.043,Z 360.333,A -85,B 0,C 180,E1 -4488.55,E2 -4488.55} C_VEL
LIN {X 0,Y 531.053,Z 360.331,A -85,B 0,C 180,E1 -4491.629,E2 -4491.629} C_VEL
LIN {X 0,Y 531.117,Z 360.326,A -85,B 0,C 180,E1 -4494.685,E2 -4494.685} C_VEL
LIN {X 0,Y 531.132,Z 360.32,A -85,B 0,C 180,E1 -4497.725,E2 -4497.725} C_VEL
LIN {X 0,Y 531.149,Z 360.324,A -85,B 0,C 180,E1 -4500.758,E2 -4500.758} C_VEL
LIN {X 0,Y 531.103,Z 360.33,A -85,B 0,C 180,E1 -4503.034,E2 -4503.034} C_VEL
LIN {X 0,Y 531.076,Z 360.327,A -85,B 0,C 180,E1 -4506.077,E2 -4506.077} C_VEL
LIN {X 0,Y 531.029,Z 360.337,A -85,B 0,C 180,E1 -4509.138,E2 -4509.138} C_VEL
LIN {X 0,Y 531.033,Z 360.334,A -85,B 0,C 180,E1 -4512.225,E2 -4512.225} C_VEL
LIN {X 0,Y 530.988,Z 360.339,A -85,B 0,C 180,E1 -4515.35,E2 -4515.35} C_VEL
LIN {X 0,Y 531.008,Z 360.335,A -85,B 0,C 180,E1 -4517.723,E2 -4517.723} C_VEL
LIN {X 0,Y 530.997,Z 360.341,A -85,B 0,C 180,E1 -4520.938,E2 -4520.938} C_VEL
LIN {X 0,Y 531,Z 360.338,A -85,B 0,C 180,E1 -4524.046,E2 -4524.046} C_VEL
LIN {X 0,Y 531.004,Z 360.342,A -85,B 0,C 180,E1 -4526.744,E2 -4526.744} C_VEL
LIN {X 0,Y 530.976,Z 360.339,A -85,B 0,C 180,E1 -4529.323,E2 -4529.323} C_VEL
LIN {X 0,Y 530.974,Z 360.343,A -85,B 0,C 180,E1 -4532.104,E2 -4532.104} C_VEL
LIN {X 0,Y 530.977,Z 360.342,A -85,B 0,C 180,E1 -4534.854,E2 -4534.854} C_VEL
LIN {X 0,Y 530.962,Z 360.341,A -85,B 0,C 180,E1 -4537.508,E2 -4537.508} C_VEL
LIN {X 0,Y 531.022,Z 360.342,A -85,B 0,C 180,E1 -4540.429,E2 -4540.429} C_VEL
LIN {X 0,Y 530.96,Z 360.341,A -85,B 0,C 180,E1 -4543.584,E2 -4543.584} C_VEL
LIN {X 0,Y 530.286,Z 360.432,A -85,B 0,C 180,E1 -4544.217,E2 -4544.217} C_VEL
LIN {X 0,Y 527.435,Z 360.786,A -85,B 0,C 180,E1 -4545.246,E2 -4545.246} C_VEL
LIN {X 0,Y 525.03,Z 361.085,A -85,B 0,C 180,E1 -4546.074,E2 -4546.074} C_VEL
LIN {X 0,Y 523.997,Z 361.212,A -85,B 0,C 180,E1 -4546.714,E2 -4546.714} C_VEL
LIN {X 0,Y 523.913,Z 361.22,A -85,B 0,C 180,E1 -4546.931,E2 -4546.931} C_VEL
LIN {X 0,Y 523.946,Z 361.219,A -85,B 0,C 180,E1 -4549.921,E2 -4549.921} C_VEL
LIN {X 0,Y 523.91,Z 361.22,A -85,B 0,C 180,E1 -4552.869,E2 -4552.869} C_VEL
LIN {X 0,Y 523.943,Z 361.218,A -85,B 0,C 180,E1 -4555.711,E2 -4555.711} C_VEL
LIN {X 0,Y 523.922,Z 361.222,A -85,B 0,C 180,E1 -4558.457,E2 -4558.457} C_VEL
LIN {X 0,Y 523.942,Z 361.215,A -85,B 0,C 180,E1 -4561.126,E2 -4561.126} C_VEL
LIN {X 0,Y 523.985,Z 361.218,A -85,B 0,C 180,E1 -4563.981,E2 -4563.981} C_VEL
LIN {X 0,Y 523.912,Z 361.222,A -85,B 0,C 180,E1 -4567.107,E2 -4567.107} C_VEL
LIN {X 0,Y 524.009,Z 361.265,A -85,B 0,C 180,E1 -4570.073,E2 -4570.073} C_VEL
LIN {X 0,Y 524.657,Z 366.914,A -85,B 0,C 180,E1 -4571.247,E2 -4571.247} C_VEL
LIN {X 0,Y 524.283,Z 382.011,A -85,B 0,C 180,E1 -4574.25,E2 -4574.25} C_VEL
LIN {X 0,Y 524.236,Z 385.413,A -85,B 0,C 180,E1 -4574.908,E2 -4574.908} C_VEL
LIN {X 0,Y 526.009,Z 395.941,A -85,B 0,C 180,E1 -4575.107,E2 -4575.107} C_VEL
LIN {X 0,Y 525.54,Z 491.992,A -85,B 0,C 180,E1 -4576.441,E2 -4576.441} C_VEL
LIN {X 0,Y 525.361,Z 505.163,A -85,B 0,C 180,E1 -4576.781,E2 -4576.781} C_VEL
LIN {X 0,Y 525.157,Z 517.252,A -85,B 0,C 180,E1 -4577.243,E2 -4577.243} C_VEL
LIN {X 0,Y 524.952,Z 527.695,A -85,B 0,C 180,E1 -4577.774,E2 -4577.774} C_VEL
LIN {X 0,Y 524.68,Z 539.032,A -85,B 0,C 180,E1 -4578.507,E2 -4578.507} C_VEL
LIN {X 0,Y 524.341,Z 549.72,A -85,B 0,C 180,E1 -4579.38,E2 -4579.38} C_VEL
LIN {X 0,Y 524.104,Z 559.33,A -85,B 0,C 180,E1 -4580.351,E2 -4580.351} C_VEL
LIN {X 0,Y 523.876,Z 567.202,A -85,B 0,C 180,E1 -4581.32,E2 -4581.32} C_VEL
LIN {X 0,Y 523.673,Z 574.898,A -85,B 0,C 180,E1 -4582.481,E2 -4582.481} C_VEL
LIN {X 0,Y 523.565,Z 581.952,A -85,B 0,C 180,E1 -4583.835,E2 -4583.835} C_VEL
LIN {X 0,Y 523.384,Z 586.658,A -85,B 0,C 180,E1 -4584.993,E2 -4584.993} C_VEL
LIN {X 0,Y 523.443,Z 590.255,A -85,B 0,C 180,E1 -4586.151,E2 -4586.151} C_VEL
LIN {X 0,Y 523.368,Z 592.119,A -85,B 0,C 180,E1 -4586.921,E2 -4586.921} C_VEL
LIN {X 0,Y 523.335,Z 593.525,A -85,B 0,C 180,E1 -4587.691,E2 -4587.691} C_VEL
LIN {X 0,Y 523.25,Z 595.141,A -85,B 0,C 180,E1 -4589.23,E2 -4589.23} C_VEL
LIN {X 0,Y 523.25,Z 595.379,A -85,B 0,C 180,E1 -4590,E2 -4590} C_VEL
LIN {X 0,Y 523.25,Z 595.196,A -85,B 0,C 180,E1 -4590.77,E2 -4590.77} C_VEL
LIN {X 0,Y 523.335,Z 593.652,A -85,B 0,C 180,E1 -4592.309,E2 -4592.309} C_VEL
LIN {X 0,Y 523.368,Z 592.301,A -85,B 0,C 180,E1 -4593.079,E2 -4593.079} C_VEL
LIN {X 0,Y 523.443,Z 589.445,A -85,B 0,C 180,E1 -4594.235,E2 -4594.235} C_VEL
LIN {X 0,Y 523.463,Z 585.574,A -85,B 0,C 180,E1 -4595.393,E2 -4595.393} C_VEL
LIN {X 0,Y 523.571,Z 580.225,A -85,B 0,C 180,E1 -4596.625,E2 -4596.625} C_VEL
LIN {X 0,Y 523.728,Z 573.067,A -85,B 0,C 180,E1 -4597.906,E2 -4597.906} C_VEL
LIN {X 0,Y 523.909,Z 564.934,A -85,B 0,C 180,E1 -4599.069,E2 -4599.069} C_VEL
LIN {X 0,Y 524.128,Z 556.607,A -85,B 0,C 180,E1 -4600.039,E2 -4600.039} C_VEL
LIN {X 0,Y 524.443,Z 546.324,A -85,B 0,C 180,E1 -4601.009,E2 -4601.009} C_VEL
LIN {X 0,Y 524.792,Z 534.912,A -85,B 0,C 180,E1 -4601.868,E2 -4601.868} C_VEL
LIN {X 0,Y 525.012,Z 524.988,A -85,B 0,C 180,E1 -4602.465,E2 -4602.465} C_VEL
LIN {X 0,Y 525.212,Z 513.692,A -85,B 0,C 180,E1 -4603.001,E2 -4603.001} C_VEL
LIN {X 0,Y 525.444,Z 500.859,A -85,B 0,C 180,E1 -4603.438,E2 -4603.438} C_VEL
LIN {X 0,Y 525.613,Z 487.197,A -85,B 0,C 180,E1 -4603.729,E2 -4603.729} C_VEL
LIN {X 0,Y 525.985,Z 395.207,A -85,B 0,C 180,E1 -4604.994,E2 -4604.994} C_VEL
LIN {X 0,Y 524.219,Z 385.306,A -85,B 0,C 180,E1 -4605.189,E2 -4605.189} C_VEL
LIN {X 0,Y 524.542,Z 371.341,A -85,B 0,C 180,E1 -4607.957,E2 -4607.957} C_VEL
LIN {X 0,Y 524.525,Z 364.357,A -85,B 0,C 180,E1 -4609.367,E2 -4609.367} C_VEL
LIN {X 0,Y 523.987,Z 361.219,A -85,B 0,C 180,E1 -4610.04,E2 -4610.04} C_VEL
LIN {X 0,Y 523.919,Z 361.224,A -85,B 0,C 180,E1 -4612.893,E2 -4612.893} C_VEL
LIN {X 0,Y 523.954,Z 361.218,A -85,B 0,C 180,E1 -4615.418,E2 -4615.418} C_VEL
LIN {X 0,Y 523.97,Z 361.221,A -85,B 0,C 180,E1 -4617.998,E2 -4617.998} C_VEL
LIN {X 0,Y 523.945,Z 361.215,A -85,B 0,C 180,E1 -4620.854,E2 -4620.854} C_VEL
LIN {X 0,Y 523.961,Z 361.219,A -85,B 0,C 180,E1 -4623.734,E2 -4623.734} C_VEL
LIN {X 0,Y 523.921,Z 361.22,A -85,B 0,C 180,E1 -4626.404,E2 -4626.404} C_VEL
LIN {X 0,Y 523.921,Z 361.218,A -85,B 0,C 180,E1 -4629.084,E2 -4629.084} C_VEL
LIN {X 0,Y 523.95,Z 361.219,A -85,B 0,C 180,E1 -4632.118,E2 -4632.118} C_VEL
LIN {X 0,Y 523.952,Z 361.217,A -85,B 0,C 180,E1 -4635.308,E2 -4635.308} C_VEL
LIN {X 0,Y 523.968,Z 361.212,A -85,B 0,C 180,E1 -4638.687,E2 -4638.687} C_VEL
LIN {X 0,Y 523.92,Z 361.22,A -85,B 0,C 180,E1 -4641.079,E2 -4641.079} C_VEL
LIN {X 0,Y 523.924,Z 361.223,A -85,B 0,C 180,E1 -4643.827,E2 -4643.827} C_VEL
LIN {X 0,Y 523.938,Z 361.216,A -85,B 0,C 180,E1 -4646.635,E2 -4646.635} C_VEL
LIN {X 0,Y 523.95,Z 361.221,A -85,B 0,C 180,E1 -4649.355,E2 -4649.355} C_VEL
LIN {X 0,Y 523.973,Z 361.212,A -85,B 0,C 180,E1 -4652.28,E2 -4652.28} C_VEL
LIN {X 0,Y 523.948,Z 361.215,A -85,B 0,C 180,E1 -4654.581,E2 -4654.581} C_VEL
LIN {X 0,Y 523.937,Z 361.22,A -85,B 0,C 180,E1 -4657.107,E2 -4657.107} C_VEL
LIN {X 0,Y 523.971,Z 361.214,A -85,B 0,C 180,E1 -4659.865,E2 -4659.865} C_VEL
LIN {X 0,Y 523.963,Z 361.215,A -85,B 0,C 180,E1 -4662.837,E2 -4662.837} C_VEL
LIN {X 0,Y 523.995,Z 361.217,A -85,B 0,C 180,E1 -4665.236,E2 -4665.236} C_VEL
LIN {X 0,Y 524.002,Z 361.208,A -85,B 0,C 180,E1 -4668.394,E2 -4668.394} C_VEL
LIN {X 0,Y 524,Z 361.213,A -85,B 0,C 180,E1 -4671.516,E2 -4671.516} C_VEL
LIN {X 0,Y 524.077,Z 361.2,A -85,B 0,C 180,E1 -4674.614,E2 -4674.614} C_VEL
LIN {X 0,Y 524.104,Z 361.197,A -85,B 0,C 180,E1 -4677.694,E2 -4677.694} C_VEL
LIN {X 0,Y 524.118,Z 361.198,A -85,B 0,C 180,E1 -4680.768,E2 -4680.768} C_VEL
LIN {X 0,Y 524.07,Z 361.209,A -85,B 0,C 180,E1 -4683.075,E2 -4683.075} C_VEL
LIN {X 0,Y 524.038,Z 361.203,A -85,B 0,C 180,E1 -4686.159,E2 -4686.159} C_VEL
LIN {X 0,Y 523.997,Z 361.213,A -85,B 0,C 180,E1 -4689.262,E2 -4689.262} C_VEL
LIN {X 0,Y 524.015,Z 361.206,A -85,B 0,C 180,E1 -4691.751,E2 -4691.751} C_VEL
LIN {X 0,Y 523.983,Z 361.217,A -85,B 0,C 180,E1 -4695.053,E2 -4695.053} C_VEL
LIN {X 0,Y 523.956,Z 361.214,A -85,B 0,C 180,E1 -4697.969,E2 -4697.969} C_VEL
LIN {X 0,Y 523.965,Z 361.216,A -85,B 0,C 180,E1 -4700.41,E2 -4700.41} C_VEL
LIN {X 0,Y 523.937,Z 361.223,A -85,B 0,C 180,E1 -4702.892,E2 -4702.892} C_VEL
LIN {X 0,Y 523.978,Z 361.211,A -85,B 0,C 180,E1 -4706.021,E2 -4706.021} C_VEL
LIN {X 0,Y 523.934,Z 361.223,A -85,B 0,C 180,E1 -4708.875,E2 -4708.875} C_VEL
LIN {X 0,Y 523.925,Z 361.217,A -85,B 0,C 180,E1 -4711.544,E2 -4711.544} C_VEL
LIN {X 0,Y 523.94,Z 361.22,A -85,B 0,C 180,E1 -4714.29,E2 -4714.29} C_VEL
LIN {X 0,Y 523.906,Z 361.222,A -85,B 0,C 180,E1 -4717.132,E2 -4717.132} C_VEL
LIN {X 0,Y 523.963,Z 361.216,A -85,B 0,C 180,E1 -4720.135,E2 -4720.135} C_VEL
LIN {X 0,Y 523.922,Z 361.219,A -85,B 0,C 180,E1 -4723.167,E2 -4723.167} C_VEL
LIN {X 0,Y 523.937,Z 361.217,A -85,B 0,C 180,E1 -4725.773,E2 -4725.773} C_VEL
LIN {X 0,Y 523.941,Z 361.218,A -85,B 0,C 180,E1 -4728.909,E2 -4728.909} C_VEL
LIN {X 0,Y 523.915,Z 361.221,A -85,B 0,C 180,E1 -4731.899,E2 -4731.899} C_VEL
LIN {X 0,Y 523.938,Z 361.217,A -85,B 0,C 180,E1 -4734.91,E2 -4734.91} C_VEL
LIN {X 0,Y 523.942,Z 361.217,A -85,B 0,C 180,E1 -4737.679,E2 -4737.679} C_VEL
LIN {X 0,Y 523.954,Z 361.219,A -85,B 0,C 180,E1 -4740.677,E2 -4740.677} C_VEL
LIN {X 0,Y 523.975,Z 361.218,A -85,B 0,C 180,E1 -4743.729,E2 -4743.729} C_VEL
LIN {X 0,Y 524.016,Z 361.335,A -85,B 0,C 180,E1 -4745.38,E2 -4745.38} C_VEL
LIN {X 0,Y 525.492,Z 369.582,A -85,B 0,C 180,E1 -4746.763,E2 -4746.763} C_VEL
LIN {X 0,Y 525.027,Z 389.246,A -85,B 0,C 180,E1 -4749.838,E2 -4749.838} C_VEL
LIN {X 0,Y 524.546,Z 408.855,A -85,B 0,C 180,E1 -4752.857,E2 -4752.857} C_VEL
LIN {X 0,Y 524.32,Z 421.85,A -85,B 0,C 180,E1 -4754.831,E2 -4754.831} C_VEL
LIN {X 0,Y 525.922,Z 432.926,A -85,B 0,C 180,E1 -4755.042,E2 -4755.042} C_VEL
LIN {X 0,Y 525.499,Z 530.237,A -85,B 0,C 180,E1 -4756.391,E2 -4756.391} C_VEL
LIN {X 0,Y 525.333,Z 543.525,A -85,B 0,C 180,E1 -4756.732,E2 -4756.732} C_VEL
LIN {X 0,Y 525.052,Z 555.701,A -85,B 0,C 180,E1 -4757.192,E2 -4757.192} C_VEL
LIN {X 0,Y 524.749,Z 568.051,A -85,B 0,C 180,E1 -4757.827,E2 -4757.827} C_VEL
LIN {X 0,Y 524.525,Z 579.607,A -85,B 0,C 180,E1 -4758.602,E2 -4758.602} C_VEL
LIN {X 0,Y 524.223,Z 590.066,A -85,B 0,C 180,E1 -4759.475,E2 -4759.475} C_VEL
LIN {X 0,Y 524,Z 598.62,A -85,B 0,C 180,E1 -4760.349,E2 -4760.349} C_VEL
LIN {X 0,Y 523.821,Z 606.515,A -85,B 0,C 180,E1 -4761.319,E2 -4761.319} C_VEL
LIN {X 0,Y 523.612,Z 614.224,A -85,B 0,C 180,E1 -4762.481,E2 -4762.481} C_VEL
LIN {X 0,Y 523.494,Z 621.334,A -85,B 0,C 180,E1 -4763.835,E2 -4763.835} C_VEL
LIN {X 0,Y 523.384,Z 626.063,A -85,B 0,C 180,E1 -4764.993,E2 -4764.993} C_VEL
LIN {X 0,Y 523.443,Z 629.681,A -85,B 0,C 180,E1 -4766.151,E2 -4766.151} C_VEL
LIN {X 0,Y 523.367,Z 631.543,A -85,B 0,C 180,E1 -4766.921,E2 -4766.921} C_VEL
LIN {X 0,Y 523.334,Z 632.94,A -85,B 0,C 180,E1 -4767.691,E2 -4767.691} C_VEL
LIN {X 0,Y 523.25,Z 634.544,A -85,B 0,C 180,E1 -4769.23,E2 -4769.23} C_VEL
LIN {X 0,Y 523.247,Z 634.761,A -85,B 0,C 180,E1 -4770,E2 -4770} C_VEL
LIN {X 0,Y 523.274,Z 633.938,A -85,B 0,C 180,E1 -4771.539,E2 -4771.539} C_VEL
LIN {X 0,Y 523.334,Z 632.943,A -85,B 0,C 180,E1 -4772.309,E2 -4772.309} C_VEL
LIN {X 0,Y 523.367,Z 631.547,A -85,B 0,C 180,E1 -4773.079,E2 -4773.079} C_VEL
LIN {X 0,Y 523.424,Z 628.608,A -85,B 0,C 180,E1 -4774.235,E2 -4774.235} C_VEL
LIN {X 0,Y 523.461,Z 624.629,A -85,B 0,C 180,E1 -4775.393,E2 -4775.393} C_VEL
LIN {X 0,Y 523.518,Z 619.391,A -85,B 0,C 180,E1 -4776.576,E2 -4776.576} C_VEL
LIN {X 0,Y 523.653,Z 613.062,A -85,B 0,C 180,E1 -4777.713,E2 -4777.713} C_VEL
LIN {X 0,Y 523.836,Z 605.021,A -85,B 0,C 180,E1 -4778.875,E2 -4778.875} C_VEL
LIN {X 0,Y 524.061,Z 596.83,A -85,B 0,C 180,E1 -4779.845,E2 -4779.845} C_VEL
LIN {X 0,Y 524.344,Z 586.844,A -85,B 0,C 180,E1 -4780.815,E2 -4780.815} C_VEL
LIN {X 0,Y 524.606,Z 575.598,A -85,B 0,C 180,E1 -4781.688,E2 -4781.688} C_VEL
LIN {X 0,Y 524.915,Z 564.531,A -85,B 0,C 180,E1 -4782.37,E2 -4782.37} C_VEL
LIN {X 0,Y 525.122,Z 552.295,A -85,B 0,C 180,E1 -4782.954,E2 -4782.954} C_VEL
LIN {X 0,Y 525.362,Z 539.474,A -85,B 0,C 180,E1 -4783.391,E2 -4783.391} C_VEL
LIN {X 0,Y 525.583,Z 525.891,A -85,B 0,C 180,E1 -4783.681,E2 -4783.681} C_VEL
LIN {X 0,Y 525.803,Z 431.605,A -85,B 0,C 180,E1 -4784.979,E2 -4784.979} C_VEL
LIN {X 0,Y 524.318,Z 421.764,A -85,B 0,C 180,E1 -4785.183,E2 -4785.183} C_VEL
LIN {X 0,Y 524.744,Z 401.27,A -85,B 0,C 180,E1 -4788.304,E2 -4788.304} C_VEL
LIN {X 0,Y 525.252,Z 381.39,A -85,B 0,C 180,E1 -4791.383,E2 -4791.383} C_VEL
